LIN {X 0,Y 712.232,Z 484.504,A -85,B 0,C 180,E1 31176.986,E2 31176.986} C_VEL
LIN {X 0,Y 712.279,Z 484.496,A -85,B 0,C 180,E1 31174.064,E2 31174.064} C_VEL
LIN {X 0,Y 712.227,Z 484.507,A -85,B 0,C 180,E1 31171.201,E2 31171.201} C_VEL
LIN {X 0,Y 712.264,Z 484.499,A -85,B 0,C 180,E1 31168.418,E2 31168.418} C_VEL
LIN {X 0,Y 712.248,Z 484.506,A -85,B 0,C 180,E1 31165.352,E2 31165.352} C_VEL
LIN {X 0,Y 712.232,Z 484.504,A -85,B 0,C 180,E1 31162.623,E2 31162.623} C_VEL
LIN {X 0,Y 712.278,Z 484.504,A -85,B 0,C 180,E1 31159.689,E2 31159.689} C_VEL
LIN {X 0,Y 712.231,Z 484.504,A -85,B 0,C 180,E1 31156.81,E2 31156.81} C_VEL
LIN {X 0,Y 712.272,Z 484.5,A -85,B 0,C 180,E1 31153.972,E2 31153.972} C_VEL
LIN {X 0,Y 712.253,Z 484.509,A -85,B 0,C 180,E1 31150.925,E2 31150.925} C_VEL
LIN {X 0,Y 712.246,Z 484.496,A -85,B 0,C 180,E1 31148.07,E2 31148.07} C_VEL
LIN {X 0,Y 712.279,Z 484.51,A -85,B 0,C 180,E1 31145.074,E2 31145.074} C_VEL
LIN {X 0,Y 712.234,Z 484.505,A -85,B 0,C 180,E1 31142.253,E2 31142.253} C_VEL
LIN {X 0,Y 712.282,Z 484.497,A -85,B 0,C 180,E1 31139.437,E2 31139.437} C_VEL
LIN {X 0,Y 712.247,Z 484.508,A -85,B 0,C 180,E1 31136.378,E2 31136.378} C_VEL
LIN {X 0,Y 712.256,Z 484.497,A -85,B 0,C 180,E1 31133.552,E2 31133.552} C_VEL
LIN {X 0,Y 712.274,Z 484.505,A -85,B 0,C 180,E1 31130.465,E2 31130.465} C_VEL
LIN {X 0,Y 712.243,Z 484.503,A -85,B 0,C 180,E1 31127.597,E2 31127.597} C_VEL
LIN {X 0,Y 712.272,Z 484.501,A -85,B 0,C 180,E1 31124.661,E2 31124.661} C_VEL
LIN {X 0,Y 712.243,Z 484.502,A -85,B 0,C 180,E1 31121.756,E2 31121.756} C_VEL
LIN {X 0,Y 712.276,Z 484.497,A -85,B 0,C 180,E1 31120.828,E2 31120.828} C_VEL
LIN {X 0,Y 711.28,Z 484.631,A -85,B 0,C 180,E1 31120.209,E2 31120.209} C_VEL
LIN {X 0,Y 704.888,Z 485.433,A -85,B 0,C 180,E1 31118.473,E2 31118.473} C_VEL
LIN {X 0,Y 704.331,Z 485.495,A -85,B 0,C 180,E1 31118.022,E2 31118.022} C_VEL
LIN {X 0,Y 704.317,Z 485.491,A -85,B 0,C 180,E1 31115.062,E2 31115.062} C_VEL
LIN {X 0,Y 704.34,Z 485.497,A -85,B 0,C 180,E1 31111.973,E2 31111.973} C_VEL
LIN {X 0,Y 704.311,Z 485.491,A -85,B 0,C 180,E1 31109.032,E2 31109.032} C_VEL
LIN {X 0,Y 704.331,Z 485.492,A -85,B 0,C 180,E1 31106.088,E2 31106.088} C_VEL
LIN {X 0,Y 704.307,Z 485.484,A -85,B 0,C 180,E1 31103.194,E2 31103.194} C_VEL
LIN {X 0,Y 704.34,Z 485.487,A -85,B 0,C 180,E1 31100.295,E2 31100.295} C_VEL
LIN {X 0,Y 704.323,Z 485.482,A -85,B 0,C 180,E1 31097.266,E2 31097.266} C_VEL
LIN {X 0,Y 704.337,Z 485.49,A -85,B 0,C 180,E1 31094.301,E2 31094.301} C_VEL
LIN {X 0,Y 704.337,Z 485.5,A -85,B 0,C 180,E1 31091.199,E2 31091.199} C_VEL
LIN {X 0,Y 704.347,Z 485.574,A -85,B 0,C 180,E1 31088.134,E2 31088.134} C_VEL
LIN {X 0,Y 704.441,Z 486.103,A -85,B 0,C 180,E1 31088.022,E2 31088.022} C_VEL
LIN {X 0,Y 711.05,Z 503.243,A -85,B 0,C 180,E1 31086.452,E2 31086.452} C_VEL
LIN {X 0,Y 710.006,Z 548.76,A -85,B 0,C 180,E1 31083.555,E2 31083.555} C_VEL
LIN {X 0,Y 708.985,Z 595.763,A -85,B 0,C 180,E1 31080.65,E2 31080.65} C_VEL
LIN {X 0,Y 708.154,Z 640.537,A -85,B 0,C 180,E1 31077.954,E2 31077.954} C_VEL
LIN {X 0,Y 708.048,Z 651.379,A -85,B 0,C 180,E1 31077.319,E2 31077.319} C_VEL
LIN {X 0,Y 709.566,Z 661.534,A -85,B 0,C 180,E1 31077.131,E2 31077.131} C_VEL
LIN {X 0,Y 708.424,Z 936.016,A -85,B 0,C 180,E1 31074.153,E2 31074.153} C_VEL
LIN {X 0,Y 708.197,Z 963.102,A -85,B 0,C 180,E1 31073.806,E2 31073.806} C_VEL
LIN {X 0,Y 707.957,Z 984.724,A -85,B 0,C 180,E1 31073.382,E2 31073.382} C_VEL
LIN {X 0,Y 707.588,Z 1005.615,A -85,B 0,C 180,E1 31072.823,E2 31072.823} C_VEL
LIN {X 0,Y 707.174,Z 1027.007,A -85,B 0,C 180,E1 31072.092,E2 31072.092} C_VEL
LIN {X 0,Y 706.746,Z 1047.449,A -85,B 0,C 180,E1 31071.234,E2 31071.234} C_VEL
LIN {X 0,Y 706.293,Z 1066.132,A -85,B 0,C 180,E1 31070.294,E2 31070.294} C_VEL
LIN {X 0,Y 705.844,Z 1084.752,A -85,B 0,C 180,E1 31069.186,E2 31069.186} C_VEL
LIN {X 0,Y 705.405,Z 1102.998,A -85,B 0,C 180,E1 31067.913,E2 31067.913} C_VEL
LIN {X 0,Y 705.047,Z 1118.673,A -85,B 0,C 180,E1 31066.646,E2 31066.646} C_VEL
LIN {X 0,Y 704.714,Z 1133.801,A -85,B 0,C 180,E1 31065.217,E2 31065.217} C_VEL
LIN {X 0,Y 704.453,Z 1147.488,A -85,B 0,C 180,E1 31063.711,E2 31063.711} C_VEL
LIN {X 0,Y 704.251,Z 1159.774,A -85,B 0,C 180,E1 31062.129,E2 31062.129} C_VEL
LIN {X 0,Y 704.113,Z 1170.11,A -85,B 0,C 180,E1 31060.555,E2 31060.555} C_VEL
LIN {X 0,Y 704.015,Z 1179.066,A -85,B 0,C 180,E1 31058.905,E2 31058.905} C_VEL
LIN {X 0,Y 703.96,Z 1186.69,A -85,B 0,C 180,E1 31057.18,E2 31057.18} C_VEL
LIN {X 0,Y 703.924,Z 1192.529,A -85,B 0,C 180,E1 31055.461,E2 31055.461} C_VEL
LIN {X 0,Y 703.914,Z 1196.698,A -85,B 0,C 180,E1 31053.746,E2 31053.746} C_VEL
LIN {X 0,Y 703.917,Z 1199.44,A -85,B 0,C 180,E1 31051.954,E2 31051.954} C_VEL
LIN {X 0,Y 703.907,Z 1200.448,A -85,B 0,C 180,E1 31050.163,E2 31050.163} C_VEL
LIN {X 0,Y 703.905,Z 1199.787,A -85,B 0,C 180,E1 31048.372,E2 31048.372} C_VEL
LIN {X 0,Y 703.906,Z 1197.502,A -85,B 0,C 180,E1 31046.58,E2 31046.58} C_VEL
LIN {X 0,Y 703.921,Z 1193.692,A -85,B 0,C 180,E1 31044.866,E2 31044.866} C_VEL
LIN {X 0,Y 703.931,Z 1188.233,A -85,B 0,C 180,E1 31043.148,E2 31043.148} C_VEL
LIN {X 0,Y 703.997,Z 1181.131,A -85,B 0,C 180,E1 31041.424,E2 31041.424} C_VEL
LIN {X 0,Y 704.079,Z 1172.545,A -85,B 0,C 180,E1 31039.775,E2 31039.775} C_VEL
LIN {X 0,Y 704.201,Z 1162.131,A -85,B 0,C 180,E1 31038.119,E2 31038.119} C_VEL
LIN {X 0,Y 704.399,Z 1150.346,A -85,B 0,C 180,E1 31036.539,E2 31036.539} C_VEL
LIN {X 0,Y 704.658,Z 1137.101,A -85,B 0,C 180,E1 31035.034,E2 31035.034} C_VEL
LIN {X 0,Y 704.954,Z 1122.438,A -85,B 0,C 180,E1 31033.606,E2 31033.606} C_VEL
LIN {X 0,Y 705.339,Z 1105.832,A -85,B 0,C 180,E1 31032.213,E2 31032.213} C_VEL
LIN {X 0,Y 705.749,Z 1088.787,A -85,B 0,C 180,E1 31030.983,E2 31030.983} C_VEL
LIN {X 0,Y 706.205,Z 1070.106,A -85,B 0,C 180,E1 31029.838,E2 31029.838} C_VEL
LIN {X 0,Y 706.666,Z 1050.479,A -85,B 0,C 180,E1 31028.82,E2 31028.82} C_VEL
LIN {X 0,Y 707.104,Z 1030.455,A -85,B 0,C 180,E1 31027.95,E2 31027.95} C_VEL
LIN {X 0,Y 707.531,Z 1009.93,A -85,B 0,C 180,E1 31027.219,E2 31027.219} C_VEL
LIN {X 0,Y 707.864,Z 988.627,A -85,B 0,C 180,E1 31026.624,E2 31026.624} C_VEL
LIN {X 0,Y 708.181,Z 965.883,A -85,B 0,C 180,E1 31026.151,E2 31026.151} C_VEL
LIN {X 0,Y 708.392,Z 943.778,A -85,B 0,C 180,E1 31025.841,E2 31025.841} C_VEL
LIN {X 0,Y 709.534,Z 668.723,A -85,B 0,C 180,E1 31022.858,E2 31022.858} C_VEL
LIN {X 0,Y 709.316,Z 658.636,A -85,B 0,C 180,E1 31022.737,E2 31022.737} C_VEL
LIN {X 0,Y 708.045,Z 651.346,A -85,B 0,C 180,E1 31022.59,E2 31022.59} C_VEL
LIN {X 0,Y 708.834,Z 604.03,A -85,B 0,C 180,E1 31019.763,E2 31019.763} C_VEL
LIN {X 0,Y 709.788,Z 557.758,A -85,B 0,C 180,E1 31016.917,E2 31016.917} C_VEL
LIN {X 0,Y 710.872,Z 510.794,A -85,B 0,C 180,E1 31013.945,E2 31013.945} C_VEL
LIN {X 0,Y 710.891,Z 502.371,A -85,B 0,C 180,E1 31013.391,E2 31013.391} C_VEL
LIN {X 0,Y 704.379,Z 485.802,A -85,B 0,C 180,E1 31011.853,E2 31011.853} C_VEL
LIN {X 0,Y 704.318,Z 485.476,A -85,B 0,C 180,E1 31010.927,E2 31010.927} C_VEL
LIN {X 0,Y 704.339,Z 485.484,A -85,B 0,C 180,E1 31007.93,E2 31007.93} C_VEL
LIN {X 0,Y 704.306,Z 485.497,A -85,B 0,C 180,E1 31004.992,E2 31004.992} C_VEL
LIN {X 0,Y 704.332,Z 485.489,A -85,B 0,C 180,E1 31002.072,E2 31002.072} C_VEL
LIN {X 0,Y 704.308,Z 485.49,A -85,B 0,C 180,E1 30999.18,E2 30999.18} C_VEL
LIN {X 0,Y 704.336,Z 485.49,A -85,B 0,C 180,E1 30996.262,E2 30996.262} C_VEL
LIN {X 0,Y 704.322,Z 485.487,A -85,B 0,C 180,E1 30993.229,E2 30993.229} C_VEL
LIN {X 0,Y 704.322,Z 485.497,A -85,B 0,C 180,E1 30990.264,E2 30990.264} C_VEL
LIN {X 0,Y 704.328,Z 485.485,A -85,B 0,C 180,E1 30987.11,E2 30987.11} C_VEL
LIN {X 0,Y 704.309,Z 485.498,A -85,B 0,C 180,E1 30984.223,E2 30984.223} C_VEL
LIN {X 0,Y 704.341,Z 485.49,A -85,B 0,C 180,E1 30981.223,E2 30981.223} C_VEL
LIN {X 0,Y 704.297,Z 485.489,A -85,B 0,C 180,E1 30978.371,E2 30978.371} C_VEL
LIN {X 0,Y 704.34,Z 485.492,A -85,B 0,C 180,E1 30975.479,E2 30975.479} C_VEL
LIN {X 0,Y 704.305,Z 485.492,A -85,B 0,C 180,E1 30972.462,E2 30972.462} C_VEL
LIN {X 0,Y 704.326,Z 485.493,A -85,B 0,C 180,E1 30969.561,E2 30969.561} C_VEL
LIN {X 0,Y 704.313,Z 485.487,A -85,B 0,C 180,E1 30966.418,E2 30966.418} C_VEL
LIN {X 0,Y 704.306,Z 485.497,A -85,B 0,C 180,E1 30963.581,E2 30963.581} C_VEL
LIN {X 0,Y 704.341,Z 485.487,A -85,B 0,C 180,E1 30960.488,E2 30960.488} C_VEL
LIN {X 0,Y 704.292,Z 485.495,A -85,B 0,C 180,E1 30957.64,E2 30957.64} C_VEL
LIN {X 0,Y 704.341,Z 485.497,A -85,B 0,C 180,E1 30954.787,E2 30954.787} C_VEL
LIN {X 0,Y 704.298,Z 485.486,A -85,B 0,C 180,E1 30951.838,E2 30951.838} C_VEL
LIN {X 0,Y 704.314,Z 485.499,A -85,B 0,C 180,E1 30949.033,E2 30949.033} C_VEL
LIN {X 0,Y 704.314,Z 485.491,A -85,B 0,C 180,E1 30945.866,E2 30945.866} C_VEL
LIN {X 0,Y 704.293,Z 485.493,A -85,B 0,C 180,E1 30943.08,E2 30943.08} C_VEL
LIN {X 0,Y 704.342,Z 485.488,A -85,B 0,C 180,E1 30940.08,E2 30940.08} C_VEL
LIN {X 0,Y 704.287,Z 485.495,A -85,B 0,C 180,E1 30937.196,E2 30937.196} C_VEL
LIN {X 0,Y 704.337,Z 485.495,A -85,B 0,C 180,E1 30934.343,E2 30934.343} C_VEL
LIN {X 0,Y 704.298,Z 485.49,A -85,B 0,C 180,E1 30931.323,E2 30931.323} C_VEL
LIN {X 0,Y 704.295,Z 485.497,A -85,B 0,C 180,E1 30928.598,E2 30928.598} C_VEL
LIN {X 0,Y 704.337,Z 485.489,A -85,B 0,C 180,E1 30925.565,E2 30925.565} C_VEL
LIN {X 0,Y 704.283,Z 485.495,A -85,B 0,C 180,E1 30922.785,E2 30922.785} C_VEL
LIN {X 0,Y 704.33,Z 485.484,A -85,B 0,C 180,E1 30919.977,E2 30919.977} C_VEL
LIN {X 0,Y 704.297,Z 485.485,A -85,B 0,C 180,E1 30916.931,E2 30916.931} C_VEL
LIN {X 0,Y 704.29,Z 485.5,A -85,B 0,C 180,E1 30914.191,E2 30914.191} C_VEL
LIN {X 0,Y 704.343,Z 485.487,A -85,B 0,C 180,E1 30911.199,E2 30911.199} C_VEL
LIN {X 0,Y 704.301,Z 485.633,A -85,B 0,C 180,E1 30908.496,E2 30908.496} C_VEL
LIN {X 0,Y 705.145,Z 488.254,A -85,B 0,C 180,E1 30908.226,E2 30908.226} C_VEL
LIN {X 0,Y 711.397,Z 503.301,A -85,B 0,C 180,E1 30906.894,E2 30906.894} C_VEL
LIN {X 0,Y 710.895,Z 527.91,A -85,B 0,C 180,E1 30905.413,E2 30905.413} C_VEL
LIN {X 0,Y 713.276,Z 540.379,A -85,B 0,C 180,E1 30905.117,E2 30905.117} C_VEL
LIN {X 0,Y 711.781,Z 796.504,A -85,B 0,C 180,E1 30902.16,E2 30902.16} C_VEL
LIN {X 0,Y 711.096,Z 919.207,A -85,B 0,C 180,E1 30900.746,E2 30900.746} C_VEL
LIN {X 0,Y 710.67,Z 944.945,A -85,B 0,C 180,E1 30900.302,E2 30900.302} C_VEL
LIN {X 0,Y 710.258,Z 966.602,A -85,B 0,C 180,E1 30899.791,E2 30899.791} C_VEL
LIN {X 0,Y 709.768,Z 990.595,A -85,B 0,C 180,E1 30899.078,E2 30899.078} C_VEL
LIN {X 0,Y 709.163,Z 1012.516,A -85,B 0,C 180,E1 30898.277,E2 30898.277} C_VEL
LIN {X 0,Y 708.561,Z 1035.191,A -85,B 0,C 180,E1 30897.297,E2 30897.297} C_VEL
LIN {X 0,Y 707.882,Z 1056.777,A -85,B 0,C 180,E1 30896.193,E2 30896.193} C_VEL
LIN {X 0,Y 707.236,Z 1077.766,A -85,B 0,C 180,E1 30894.961,E2 30894.961} C_VEL
LIN {X 0,Y 706.625,Z 1097.064,A -85,B 0,C 180,E1 30893.65,E2 30893.65} C_VEL
LIN {X 0,Y 706.064,Z 1115.772,A -85,B 0,C 180,E1 30892.216,E2 30892.216} C_VEL
LIN {X 0,Y 705.557,Z 1132.805,A -85,B 0,C 180,E1 30890.718,E2 30890.718} C_VEL
LIN {X 0,Y 705.141,Z 1148.973,A -85,B 0,C 180,E1 30889.12,E2 30889.12} C_VEL
LIN {X 0,Y 704.767,Z 1163.229,A -85,B 0,C 180,E1 30887.504,E2 30887.504} C_VEL
LIN {X 0,Y 704.49,Z 1177.065,A -85,B 0,C 180,E1 30885.728,E2 30885.728} C_VEL
LIN {X 0,Y 704.267,Z 1188.801,A -85,B 0,C 180,E1 30883.966,E2 30883.966} C_VEL
LIN {X 0,Y 704.115,Z 1198.949,A -85,B 0,C 180,E1 30882.215,E2 30882.215} C_VEL
LIN {X 0,Y 704.003,Z 1208.54,A -85,B 0,C 180,E1 30880.226,E2 30880.226} C_VEL
LIN {X 0,Y 703.953,Z 1215.121,A -85,B 0,C 180,E1 30878.577,E2 30878.577} C_VEL
LIN {X 0,Y 703.926,Z 1221.452,A -85,B 0,C 180,E1 30876.607,E2 30876.607} C_VEL
LIN {X 0,Y 703.911,Z 1225.814,A -85,B 0,C 180,E1 30874.726,E2 30874.726} C_VEL
LIN {X 0,Y 703.882,Z 1228.685,A -85,B 0,C 180,E1 30872.931,E2 30872.931} C_VEL
LIN {X 0,Y 703.892,Z 1230.262,A -85,B 0,C 180,E1 30870.895,E2 30870.895} C_VEL
LIN {X 0,Y 703.884,Z 1230.306,A -85,B 0,C 180,E1 30869.267,E2 30869.267} C_VEL
LIN {X 0,Y 703.886,Z 1229.017,A -85,B 0,C 180,E1 30867.313,E2 30867.313} C_VEL
LIN {X 0,Y 703.916,Z 1225.973,A -85,B 0,C 180,E1 30865.356,E2 30865.356} C_VEL
LIN {X 0,Y 703.925,Z 1221.865,A -85,B 0,C 180,E1 30863.557,E2 30863.557} C_VEL
LIN {X 0,Y 703.956,Z 1215.424,A -85,B 0,C 180,E1 30861.505,E2 30861.505} C_VEL
LIN {X 0,Y 703.996,Z 1208.765,A -85,B 0,C 180,E1 30859.826,E2 30859.826} C_VEL
LIN {X 0,Y 704.106,Z 1199.868,A -85,B 0,C 180,E1 30857.951,E2 30857.951} C_VEL
LIN {X 0,Y 704.26,Z 1189.323,A -85,B 0,C 180,E1 30856.117,E2 30856.117} C_VEL
LIN {X 0,Y 704.473,Z 1177.647,A -85,B 0,C 180,E1 30854.356,E2 30854.356} C_VEL
LIN {X 0,Y 704.749,Z 1163.936,A -85,B 0,C 180,E1 30852.581,E2 30852.581} C_VEL
LIN {X 0,Y 705.119,Z 1149.75,A -85,B 0,C 180,E1 30850.965,E2 30850.965} C_VEL
LIN {X 0,Y 705.54,Z 1133.398,A -85,B 0,C 180,E1 30849.337,E2 30849.337} C_VEL
LIN {X 0,Y 706.035,Z 1116.552,A -85,B 0,C 180,E1 30847.85,E2 30847.85} C_VEL
LIN {X 0,Y 706.604,Z 1097.667,A -85,B 0,C 180,E1 30846.394,E2 30846.394} C_VEL
LIN {X 0,Y 707.213,Z 1078.429,A -85,B 0,C 180,E1 30845.083,E2 30845.083} C_VEL
LIN {X 0,Y 707.852,Z 1057.575,A -85,B 0,C 180,E1 30843.851,E2 30843.851} C_VEL
LIN {X 0,Y 708.498,Z 1036.993,A -85,B 0,C 180,E1 30842.791,E2 30842.791} C_VEL
LIN {X 0,Y 709.128,Z 1013.638,A -85,B 0,C 180,E1 30841.768,E2 30841.768} C_VEL
LIN {X 0,Y 709.724,Z 991.879,A -85,B 0,C 180,E1 30840.966,E2 30840.966} C_VEL
LIN {X 0,Y 710.256,Z 966.819,A -85,B 0,C 180,E1 30840.214,E2 30840.214} C_VEL
LIN {X 0,Y 710.662,Z 945.208,A -85,B 0,C 180,E1 30839.704,E2 30839.704} C_VEL
LIN {X 0,Y 711.094,Z 919.454,A -85,B 0,C 180,E1 30839.258,E2 30839.258} C_VEL
LIN {X 0,Y 711.703,Z 811.771,A -85,B 0,C 180,E1 30838.014,E2 30838.014} C_VEL
LIN {X 0,Y 713.129,Z 564.423,A -85,B 0,C 180,E1 30835.164,E2 30835.164} C_VEL
LIN {X 0,Y 713.107,Z 538.54,A -85,B 0,C 180,E1 30834.851,E2 30834.851} C_VEL
LIN {X 0,Y 710.908,Z 527.965,A -85,B 0,C 180,E1 30834.588,E2 30834.588} C_VEL
LIN {X 0,Y 711.397,Z 503.3,A -85,B 0,C 180,E1 30833.106,E2 30833.106} C_VEL
LIN {X 0,Y 704.326,Z 485.803,A -85,B 0,C 180,E1 30831.541,E2 30831.541} C_VEL
LIN {X 0,Y 704.342,Z 485.485,A -85,B 0,C 180,E1 30830.558,E2 30830.558} C_VEL
LIN {X 0,Y 704.281,Z 485.485,A -85,B 0,C 180,E1 30827.705,E2 30827.705} C_VEL
LIN {X 0,Y 704.312,Z 485.494,A -85,B 0,C 180,E1 30824.991,E2 30824.991} C_VEL
LIN {X 0,Y 704.307,Z 485.5,A -85,B 0,C 180,E1 30821.855,E2 30821.855} C_VEL
LIN {X 0,Y 704.284,Z 485.478,A -85,B 0,C 180,E1 30819.182,E2 30819.182} C_VEL
LIN {X 0,Y 704.341,Z 485.495,A -85,B 0,C 180,E1 30816.263,E2 30816.263} C_VEL
LIN {X 0,Y 704.289,Z 485.482,A -85,B 0,C 180,E1 30813.328,E2 30813.328} C_VEL
LIN {X 0,Y 704.317,Z 485.491,A -85,B 0,C 180,E1 30810.547,E2 30810.547} C_VEL
LIN {X 0,Y 704.315,Z 485.5,A -85,B 0,C 180,E1 30807.469,E2 30807.469} C_VEL
LIN {X 0,Y 704.294,Z 485.489,A -85,B 0,C 180,E1 30804.67,E2 30804.67} C_VEL
LIN {X 0,Y 704.341,Z 485.496,A -85,B 0,C 180,E1 30801.748,E2 30801.748} C_VEL
LIN {X 0,Y 704.292,Z 485.496,A -85,B 0,C 180,E1 30798.887,E2 30798.887} C_VEL
LIN {X 0,Y 704.33,Z 485.486,A -85,B 0,C 180,E1 30796.042,E2 30796.042} C_VEL
LIN {X 0,Y 704.311,Z 485.493,A -85,B 0,C 180,E1 30792.962,E2 30792.962} C_VEL
LIN {X 0,Y 704.306,Z 485.491,A -85,B 0,C 180,E1 30790.139,E2 30790.139} C_VEL
LIN {X 0,Y 704.343,Z 485.493,A -85,B 0,C 180,E1 30787.095,E2 30787.095} C_VEL
LIN {X 0,Y 704.295,Z 485.489,A -85,B 0,C 180,E1 30784.234,E2 30784.234} C_VEL
LIN {X 0,Y 704.34,Z 485.49,A -85,B 0,C 180,E1 30781.383,E2 30781.383} C_VEL
LIN {X 0,Y 704.309,Z 485.496,A -85,B 0,C 180,E1 30778.454,E2 30778.454} C_VEL
LIN {X 0,Y 704.319,Z 485.489,A -85,B 0,C 180,E1 30775.603,E2 30775.603} C_VEL
LIN {X 0,Y 704.333,Z 485.5,A -85,B 0,C 180,E1 30772.495,E2 30772.495} C_VEL
LIN {X 0,Y 704.306,Z 485.485,A -85,B 0,C 180,E1 30769.613,E2 30769.613} C_VEL
LIN {X 0,Y 704.337,Z 485.497,A -85,B 0,C 180,E1 30766.621,E2 30766.621} C_VEL
LIN {X 0,Y 704.301,Z 485.495,A -85,B 0,C 180,E1 30763.759,E2 30763.759} C_VEL
LIN {X 0,Y 704.339,Z 485.485,A -85,B 0,C 180,E1 30760.857,E2 30760.857} C_VEL
LIN {X 0,Y 704.331,Z 485.495,A -85,B 0,C 180,E1 30758.022,E2 30758.022} C_VEL
LIN {X 0,Y 703.303,Z 485.614,A -85,B 0,C 180,E1 30757.395,E2 30757.395} C_VEL
LIN {X 0,Y 696.884,Z 486.424,A -85,B 0,C 180,E1 30755.639,E2 30755.639} C_VEL
LIN {X 0,Y 696.37,Z 486.481,A -85,B 0,C 180,E1 30755.183,E2 30755.183} C_VEL
LIN {X 0,Y 696.396,Z 486.481,A -85,B 0,C 180,E1 30752.181,E2 30752.181} C_VEL
LIN {X 0,Y 696.368,Z 486.484,A -85,B 0,C 180,E1 30749.323,E2 30749.323} C_VEL
LIN {X 0,Y 696.398,Z 486.476,A -85,B 0,C 180,E1 30746.381,E2 30746.381} C_VEL
LIN {X 0,Y 696.378,Z 486.473,A -85,B 0,C 180,E1 30743.38,E2 30743.38} C_VEL
LIN {X 0,Y 696.402,Z 486.475,A -85,B 0,C 180,E1 30740.395,E2 30740.395} C_VEL
LIN {X 0,Y 696.389,Z 486.468,A -85,B 0,C 180,E1 30737.317,E2 30737.317} C_VEL
LIN {X 0,Y 696.4,Z 486.479,A -85,B 0,C 180,E1 30734.249,E2 30734.249} C_VEL
LIN {X 0,Y 696.391,Z 486.489,A -85,B 0,C 180,E1 30731.116,E2 30731.116} C_VEL
LIN {X 0,Y 696.399,Z 486.668,A -85,B 0,C 180,E1 30728.527,E2 30728.527} C_VEL
LIN {X 0,Y 700.012,Z 495.946,A -85,B 0,C 180,E1 30727.623,E2 30727.623} C_VEL
LIN {X 0,Y 704.1,Z 506.677,A -85,B 0,C 180,E1 30726.644,E2 30726.644} C_VEL
LIN {X 0,Y 702.908,Z 551.847,A -85,B 0,C 180,E1 30723.743,E2 30723.743} C_VEL
LIN {X 0,Y 701.724,Z 599.512,A -85,B 0,C 180,E1 30720.771,E2 30720.771} C_VEL
LIN {X 0,Y 700.761,Z 644.343,A -85,B 0,C 180,E1 30718.043,E2 30718.043} C_VEL
LIN {X 0,Y 700.767,Z 651.94,A -85,B 0,C 180,E1 30717.615,E2 30717.615} C_VEL
LIN {X 0,Y 702.441,Z 662.731,A -85,B 0,C 180,E1 30717.416,E2 30717.416} C_VEL
LIN {X 0,Y 701.12,Z 937.085,A -85,B 0,C 180,E1 30714.409,E2 30714.409} C_VEL
LIN {X 0,Y 700.865,Z 963.369,A -85,B 0,C 180,E1 30714.067,E2 30714.067} C_VEL
LIN {X 0,Y 700.585,Z 984.94,A -85,B 0,C 180,E1 30713.638,E2 30713.638} C_VEL
LIN {X 0,Y 700.158,Z 1006.371,A -85,B 0,C 180,E1 30713.057,E2 30713.057} C_VEL
LIN {X 0,Y 699.698,Z 1027.018,A -85,B 0,C 180,E1 30712.34,E2 30712.34} C_VEL
LIN {X 0,Y 699.197,Z 1047.457,A -85,B 0,C 180,E1 30711.474,E2 30711.474} C_VEL
LIN {X 0,Y 698.68,Z 1066.146,A -85,B 0,C 180,E1 30710.525,E2 30710.525} C_VEL
LIN {X 0,Y 698.165,Z 1084.759,A -85,B 0,C 180,E1 30709.405,E2 30709.405} C_VEL
LIN {X 0,Y 697.651,Z 1103.003,A -85,B 0,C 180,E1 30708.119,E2 30708.119} C_VEL
LIN {X 0,Y 697.233,Z 1118.679,A -85,B 0,C 180,E1 30706.838,E2 30706.838} C_VEL
LIN {X 0,Y 696.845,Z 1134.062,A -85,B 0,C 180,E1 30705.367,E2 30705.367} C_VEL
LIN {X 0,Y 696.548,Z 1147.492,A -85,B 0,C 180,E1 30703.87,E2 30703.87} C_VEL
LIN {X 0,Y 696.313,Z 1159.779,A -85,B 0,C 180,E1 30702.27,E2 30702.27} C_VEL
LIN {X 0,Y 696.145,Z 1170.112,A -85,B 0,C 180,E1 30700.677,E2 30700.677} C_VEL
LIN {X 0,Y 696.03,Z 1179.069,A -85,B 0,C 180,E1 30699.008,E2 30699.008} C_VEL
LIN {X 0,Y 695.967,Z 1186.692,A -85,B 0,C 180,E1 30697.263,E2 30697.263} C_VEL
LIN {X 0,Y 695.923,Z 1192.531,A -85,B 0,C 180,E1 30695.524,E2 30695.524} C_VEL
LIN {X 0,Y 695.915,Z 1196.699,A -85,B 0,C 180,E1 30693.789,E2 30693.789} C_VEL
LIN {X 0,Y 695.917,Z 1199.44,A -85,B 0,C 180,E1 30691.976,E2 30691.976} C_VEL
LIN {X 0,Y 695.907,Z 1200.448,A -85,B 0,C 180,E1 30690.165,E2 30690.165} C_VEL
LIN {X 0,Y 695.906,Z 1199.787,A -85,B 0,C 180,E1 30688.353,E2 30688.353} C_VEL
LIN {X 0,Y 695.909,Z 1197.501,A -85,B 0,C 180,E1 30686.54,E2 30686.54} C_VEL
LIN {X 0,Y 695.924,Z 1193.69,A -85,B 0,C 180,E1 30684.807,E2 30684.807} C_VEL
LIN {X 0,Y 695.94,Z 1188.232,A -85,B 0,C 180,E1 30683.069,E2 30683.069} C_VEL
LIN {X 0,Y 696.011,Z 1181.129,A -85,B 0,C 180,E1 30681.325,E2 30681.325} C_VEL
LIN {X 0,Y 696.11,Z 1172.543,A -85,B 0,C 180,E1 30679.657,E2 30679.657} C_VEL
LIN {X 0,Y 696.261,Z 1161.937,A -85,B 0,C 180,E1 30677.954,E2 30677.954} C_VEL
LIN {X 0,Y 696.484,Z 1150.341,A -85,B 0,C 180,E1 30676.383,E2 30676.383} C_VEL
LIN {X 0,Y 696.783,Z 1137.097,A -85,B 0,C 180,E1 30674.861,E2 30674.861} C_VEL
LIN {X 0,Y 697.134,Z 1122.431,A -85,B 0,C 180,E1 30673.416,E2 30673.416} C_VEL
LIN {X 0,Y 697.579,Z 1105.826,A -85,B 0,C 180,E1 30672.008,E2 30672.008} C_VEL
LIN {X 0,Y 698.052,Z 1088.782,A -85,B 0,C 180,E1 30670.765,E2 30670.765} C_VEL
LIN {X 0,Y 698.558,Z 1070.703,A -85,B 0,C 180,E1 30669.644,E2 30669.644} C_VEL
LIN {X 0,Y 699.095,Z 1051.047,A -85,B 0,C 180,E1 30668.608,E2 30668.608} C_VEL
LIN {X 0,Y 699.593,Z 1031.566,A -85,B 0,C 180,E1 30667.745,E2 30667.745} C_VEL
LIN {X 0,Y 700.066,Z 1011.197,A -85,B 0,C 180,E1 30667.007,E2 30667.007} C_VEL
LIN {X 0,Y 700.47,Z 989.6,A -85,B 0,C 180,E1 30666.388,E2 30666.388} C_VEL
LIN {X 0,Y 700.836,Z 967.551,A -85,B 0,C 180,E1 30665.914,E2 30665.914} C_VEL
LIN {X 0,Y 701.068,Z 945.826,A -85,B 0,C 180,E1 30665.597,E2 30665.597} C_VEL
LIN {X 0,Y 702.393,Z 672.108,A -85,B 0,C 180,E1 30662.598,E2 30662.598} C_VEL
LIN {X 0,Y 702.203,Z 659.929,A -85,B 0,C 180,E1 30662.452,E2 30662.452} C_VEL
LIN {X 0,Y 700.694,Z 651.352,A -85,B 0,C 180,E1 30662.278,E2 30662.278} C_VEL
LIN {X 0,Y 701.612,Z 604.826,A -85,B 0,C 180,E1 30659.466,E2 30659.466} C_VEL
LIN {X 0,Y 702.741,Z 557.792,A -85,B 0,C 180,E1 30656.542,E2 30656.542} C_VEL
LIN {X 0,Y 703.968,Z 511.51,A -85,B 0,C 180,E1 30653.581,E2 30653.581} C_VEL
LIN {X 0,Y 704.051,Z 506.113,A -85,B 0,C 180,E1 30653.225,E2 30653.225} C_VEL
LIN {X 0,Y 696.401,Z 486.723,A -85,B 0,C 180,E1 30651.39,E2 30651.39} C_VEL
LIN {X 0,Y 696.39,Z 486.49,A -85,B 0,C 180,E1 30648.775,E2 30648.775} C_VEL
LIN {X 0,Y 696.391,Z 486.48,A -85,B 0,C 180,E1 30645.636,E2 30645.636} C_VEL
LIN {X 0,Y 696.38,Z 486.469,A -85,B 0,C 180,E1 30642.666,E2 30642.666} C_VEL
LIN {X 0,Y 696.399,Z 486.476,A -85,B 0,C 180,E1 30639.556,E2 30639.556} C_VEL
LIN {X 0,Y 696.372,Z 486.473,A -85,B 0,C 180,E1 30636.576,E2 30636.576} C_VEL
LIN {X 0,Y 696.402,Z 486.476,A -85,B 0,C 180,E1 30633.558,E2 30633.558} C_VEL
LIN {X 0,Y 696.363,Z 486.484,A -85,B 0,C 180,E1 30630.646,E2 30630.646} C_VEL
LIN {X 0,Y 696.4,Z 486.482,A -85,B 0,C 180,E1 30627.816,E2 30627.816} C_VEL
LIN {X 0,Y 696.366,Z 486.482,A -85,B 0,C 180,E1 30624.789,E2 30624.789} C_VEL
LIN {X 0,Y 696.401,Z 486.484,A -85,B 0,C 180,E1 30621.831,E2 30621.831} C_VEL
LIN {X 0,Y 696.376,Z 486.474,A -85,B 0,C 180,E1 30618.762,E2 30618.762} C_VEL
LIN {X 0,Y 696.38,Z 486.488,A -85,B 0,C 180,E1 30615.832,E2 30615.832} C_VEL
LIN {X 0,Y 696.386,Z 486.479,A -85,B 0,C 180,E1 30612.69,E2 30612.69} C_VEL
LIN {X 0,Y 696.364,Z 486.479,A -85,B 0,C 180,E1 30609.838,E2 30609.838} C_VEL
LIN {X 0,Y 696.401,Z 486.475,A -85,B 0,C 180,E1 30606.844,E2 30606.844} C_VEL
LIN {X 0,Y 696.354,Z 486.483,A -85,B 0,C 180,E1 30603.952,E2 30603.952} C_VEL
LIN {X 0,Y 696.404,Z 486.48,A -85,B 0,C 180,E1 30601.07,E2 30601.07} C_VEL
LIN {X 0,Y 696.367,Z 486.48,A -85,B 0,C 180,E1 30598.107,E2 30598.107} C_VEL
LIN {X 0,Y 696.368,Z 486.482,A -85,B 0,C 180,E1 30595.305,E2 30595.305} C_VEL
LIN {X 0,Y 696.391,Z 486.471,A -85,B 0,C 180,E1 30592.171,E2 30592.171} C_VEL
LIN {X 0,Y 696.355,Z 486.486,A -85,B 0,C 180,E1 30589.325,E2 30589.325} C_VEL
LIN {X 0,Y 696.401,Z 486.483,A -85,B 0,C 180,E1 30586.381,E2 30586.381} C_VEL
LIN {X 0,Y 696.351,Z 486.479,A -85,B 0,C 180,E1 30583.482,E2 30583.482} C_VEL
LIN {X 0,Y 696.39,Z 486.489,A -85,B 0,C 180,E1 30580.629,E2 30580.629} C_VEL
LIN {X 0,Y 696.365,Z 486.481,A -85,B 0,C 180,E1 30577.546,E2 30577.546} C_VEL
LIN {X 0,Y 696.358,Z 486.482,A -85,B 0,C 180,E1 30574.757,E2 30574.757} C_VEL
LIN {X 0,Y 696.397,Z 486.476,A -85,B 0,C 180,E1 30571.657,E2 30571.657} C_VEL
LIN {X 0,Y 696.347,Z 486.484,A -85,B 0,C 180,E1 30568.845,E2 30568.845} C_VEL
LIN {X 0,Y 696.401,Z 486.469,A -85,B 0,C 180,E1 30565.937,E2 30565.937} C_VEL
LIN {X 0,Y 696.352,Z 486.483,A -85,B 0,C 180,E1 30562.971,E2 30562.971} C_VEL
LIN {X 0,Y 696.357,Z 486.468,A -85,B 0,C 180,E1 30560.285,E2 30560.285} C_VEL
LIN {X 0,Y 696.386,Z 486.471,A -85,B 0,C 180,E1 30557.196,E2 30557.196} C_VEL
LIN {X 0,Y 696.344,Z 486.488,A -85,B 0,C 180,E1 30554.368,E2 30554.368} C_VEL
LIN {X 0,Y 696.403,Z 486.469,A -85,B 0,C 180,E1 30551.443,E2 30551.443} C_VEL
LIN {X 0,Y 696.403,Z 486.623,A -85,B 0,C 180,E1 30548.939,E2 30548.939} C_VEL
LIN {X 0,Y 697.498,Z 489.736,A -85,B 0,C 180,E1 30548.622,E2 30548.622} C_VEL
LIN {X 0,Y 704.529,Z 506.76,A -85,B 0,C 180,E1 30547.096,E2 30547.096} C_VEL
LIN {X 0,Y 704.075,Z 528.398,A -85,B 0,C 180,E1 30545.798,E2 30545.798} C_VEL
LIN {X 0,Y 706.716,Z 541.979,A -85,B 0,C 180,E1 30545.473,E2 30545.473} C_VEL
LIN {X 0,Y 704.999,Z 797.522,A -85,B 0,C 180,E1 30542.495,E2 30542.495} C_VEL
LIN {X 0,Y 704.211,Z 919.325,A -85,B 0,C 180,E1 30541.078,E2 30541.078} C_VEL
LIN {X 0,Y 703.739,Z 944.943,A -85,B 0,C 180,E1 30540.632,E2 30540.632} C_VEL
LIN {X 0,Y 703.251,Z 966.713,A -85,B 0,C 180,E1 30540.116,E2 30540.116} C_VEL
LIN {X 0,Y 702.691,Z 990.591,A -85,B 0,C 180,E1 30539.4,E2 30539.4} C_VEL
LIN {X 0,Y 702.01,Z 1012.515,A -85,B 0,C 180,E1 30538.591,E2 30538.591} C_VEL
LIN {X 0,Y 701.294,Z 1035.187,A -85,B 0,C 180,E1 30537.604,E2 30537.604} C_VEL
LIN {X 0,Y 700.539,Z 1056.573,A -85,B 0,C 180,E1 30536.5,E2 30536.5} C_VEL
LIN {X 0,Y 699.774,Z 1077.76,A -85,B 0,C 180,E1 30535.246,E2 30535.246} C_VEL
LIN {X 0,Y 699.093,Z 1096.755,A -85,B 0,C 180,E1 30533.943,E2 30533.943} C_VEL
LIN {X 0,Y 698.419,Z 1115.771,A -85,B 0,C 180,E1 30532.472,E2 30532.472} C_VEL
LIN {X 0,Y 697.846,Z 1132.471,A -85,B 0,C 180,E1 30530.989,E2 30530.989} C_VEL
LIN {X 0,Y 697.345,Z 1148.975,A -85,B 0,C 180,E1 30529.342,E2 30529.342} C_VEL
LIN {X 0,Y 696.901,Z 1163.938,A -85,B 0,C 180,E1 30527.621,E2 30527.621} C_VEL
LIN {X 0,Y 696.576,Z 1177.648,A -85,B 0,C 180,E1 30525.826,E2 30525.826} C_VEL
LIN {X 0,Y 696.321,Z 1189.322,A -85,B 0,C 180,E1 30524.044,E2 30524.044} C_VEL
LIN {X 0,Y 696.136,Z 1200.301,A -85,B 0,C 180,E1 30522.105,E2 30522.105} C_VEL
LIN {X 0,Y 696.017,Z 1208.98,A -85,B 0,C 180,E1 30520.241,E2 30520.241} C_VEL
LIN {X 0,Y 695.963,Z 1215.728,A -85,B 0,C 180,E1 30518.51,E2 30518.51} C_VEL
LIN {X 0,Y 695.927,Z 1222.071,A -85,B 0,C 180,E1 30516.434,E2 30516.434} C_VEL
LIN {X 0,Y 695.913,Z 1225.973,A -85,B 0,C 180,E1 30514.697,E2 30514.697} C_VEL
LIN {X 0,Y 695.883,Z 1228.91,A -85,B 0,C 180,E1 30512.8,E2 30512.8} C_VEL
LIN {X 0,Y 695.888,Z 1230.284,A -85,B 0,C 180,E1 30510.823,E2 30510.823} C_VEL
LIN {X 0,Y 695.888,Z 1230.284,A -85,B 0,C 180,E1 30509.177,E2 30509.177} C_VEL
LIN {X 0,Y 695.883,Z 1228.91,A -85,B 0,C 180,E1 30507.2,E2 30507.2} C_VEL
LIN {X 0,Y 695.913,Z 1225.973,A -85,B 0,C 180,E1 30505.302,E2 30505.302} C_VEL
LIN {X 0,Y 695.928,Z 1221.864,A -85,B 0,C 180,E1 30503.483,E2 30503.483} C_VEL
LIN {X 0,Y 695.96,Z 1215.424,A -85,B 0,C 180,E1 30501.407,E2 30501.407} C_VEL
LIN {X 0,Y 696.02,Z 1208.895,A -85,B 0,C 180,E1 30499.739,E2 30499.739} C_VEL
LIN {X 0,Y 696.143,Z 1199.866,A -85,B 0,C 180,E1 30497.811,E2 30497.811} C_VEL
LIN {X 0,Y 696.321,Z 1189.324,A -85,B 0,C 180,E1 30495.956,E2 30495.956} C_VEL
LIN {X 0,Y 696.593,Z 1177.122,A -85,B 0,C 180,E1 30494.096,E2 30494.096} C_VEL
LIN {X 0,Y 696.923,Z 1163.231,A -85,B 0,C 180,E1 30492.293,E2 30492.293} C_VEL
LIN {X 0,Y 697.369,Z 1148.181,A -85,B 0,C 180,E1 30490.571,E2 30490.571} C_VEL
LIN {X 0,Y 697.875,Z 1131.542,A -85,B 0,C 180,E1 30488.924,E2 30488.924} C_VEL
LIN {X 0,Y 698.487,Z 1113.618,A -85,B 0,C 180,E1 30487.352,E2 30487.352} C_VEL
LIN {X 0,Y 699.129,Z 1095.654,A -85,B 0,C 180,E1 30485.977,E2 30485.977} C_VEL
LIN {X 0,Y 699.843,Z 1075.64,A -85,B 0,C 180,E1 30484.621,E2 30484.621} C_VEL
LIN {X 0,Y 700.56,Z 1055.965,A -85,B 0,C 180,E1 30483.467,E2 30483.467} C_VEL
LIN {X 0,Y 701.325,Z 1034.264,A -85,B 0,C 180,E1 30482.351,E2 30482.351} C_VEL
LIN {X 0,Y 702.011,Z 1012.517,A -85,B 0,C 180,E1 30481.409,E2 30481.409} C_VEL
LIN {X 0,Y 702.717,Z 989.858,A -85,B 0,C 180,E1 30480.575,E2 30480.575} C_VEL
LIN {X 0,Y 703.267,Z 965.653,A -85,B 0,C 180,E1 30479.856,E2 30479.856} C_VEL
LIN {X 0,Y 703.791,Z 943.382,A -85,B 0,C 180,E1 30479.335,E2 30479.335} C_VEL
LIN {X 0,Y 704.219,Z 918.029,A -85,B 0,C 180,E1 30478.904,E2 30478.904} C_VEL
LIN {X 0,Y 705.855,Z 661.925,A -85,B 0,C 180,E1 30475.933,E2 30475.933} C_VEL
LIN {X 0,Y 706.555,Z 540.21,A -85,B 0,C 180,E1 30474.496,E2 30474.496} C_VEL
LIN {X 0,Y 704.009,Z 527.936,A -85,B 0,C 180,E1 30474.187,E2 30474.187} C_VEL
LIN {X 0,Y 704.529,Z 506.741,A -85,B 0,C 180,E1 30472.903,E2 30472.903} C_VEL
LIN {X 0,Y 696.424,Z 486.787,A -85,B 0,C 180,E1 30471.094,E2 30471.094} C_VEL
LIN {X 0,Y 696.384,Z 486.478,A -85,B 0,C 180,E1 30470.288,E2 30470.288} C_VEL
LIN {X 0,Y 696.341,Z 486.473,A -85,B 0,C 180,E1 30467.557,E2 30467.557} C_VEL
LIN {X 0,Y 696.4,Z 486.476,A -85,B 0,C 180,E1 30464.708,E2 30464.708} C_VEL
LIN {X 0,Y 696.352,Z 486.489,A -85,B 0,C 180,E1 30461.669,E2 30461.669} C_VEL
LIN {X 0,Y 696.362,Z 486.462,A -85,B 0,C 180,E1 30458.902,E2 30458.902} C_VEL
LIN {X 0,Y 696.378,Z 486.485,A -85,B 0,C 180,E1 30455.76,E2 30455.76} C_VEL
LIN {X 0,Y 696.349,Z 486.467,A -85,B 0,C 180,E1 30452.971,E2 30452.971} C_VEL
LIN {X 0,Y 696.404,Z 486.484,A -85,B 0,C 180,E1 30450.031,E2 30450.031} C_VEL
LIN {X 0,Y 696.355,Z 486.486,A -85,B 0,C 180,E1 30447.169,E2 30447.169} C_VEL
LIN {X 0,Y 696.384,Z 486.475,A -85,B 0,C 180,E1 30444.336,E2 30444.336} C_VEL
LIN {X 0,Y 696.37,Z 486.483,A -85,B 0,C 180,E1 30441.213,E2 30441.213} C_VEL
LIN {X 0,Y 696.365,Z 486.481,A -85,B 0,C 180,E1 30438.364,E2 30438.364} C_VEL
LIN {X 0,Y 696.395,Z 486.489,A -85,B 0,C 180,E1 30435.241,E2 30435.241} C_VEL
LIN {X 0,Y 696.355,Z 486.477,A -85,B 0,C 180,E1 30432.438,E2 30432.438} C_VEL
LIN {X 0,Y 696.399,Z 486.482,A -85,B 0,C 180,E1 30429.504,E2 30429.504} C_VEL
LIN {X 0,Y 696.361,Z 486.485,A -85,B 0,C 180,E1 30426.596,E2 30426.596} C_VEL
LIN {X 0,Y 696.391,Z 486.473,A -85,B 0,C 180,E1 30423.705,E2 30423.705} C_VEL
LIN {X 0,Y 696.375,Z 486.484,A -85,B 0,C 180,E1 30420.576,E2 30420.576} C_VEL
LIN {X 0,Y 696.376,Z 486.477,A -85,B 0,C 180,E1 30417.696,E2 30417.696} C_VEL
LIN {X 0,Y 696.392,Z 486.481,A -85,B 0,C 180,E1 30414.562,E2 30414.562} C_VEL
LIN {X 0,Y 696.368,Z 486.481,A -85,B 0,C 180,E1 30411.661,E2 30411.661} C_VEL
LIN {X 0,Y 696.399,Z 486.479,A -85,B 0,C 180,E1 30408.656,E2 30408.656} C_VEL
LIN {X 0,Y 696.36,Z 486.477,A -85,B 0,C 180,E1 30405.739,E2 30405.739} C_VEL
LIN {X 0,Y 696.4,Z 486.479,A -85,B 0,C 180,E1 30402.882,E2 30402.882} C_VEL
LIN {X 0,Y 696.372,Z 486.486,A -85,B 0,C 180,E1 30399.842,E2 30399.842} C_VEL
LIN {X 0,Y 696.397,Z 486.472,A -85,B 0,C 180,E1 30396.922,E2 30396.922} C_VEL
LIN {X 0,Y 696.37,Z 486.481,A -85,B 0,C 180,E1 30395.183,E2 30395.183} C_VEL
LIN {X 0,Y 695.404,Z 486.605,A -85,B 0,C 180,E1 30394.549,E2 30394.549} C_VEL
LIN {X 0,Y 688.991,Z 487.397,A -85,B 0,C 180,E1 30392.773,E2 30392.773} C_VEL
LIN {X 0,Y 688.455,Z 487.468,A -85,B 0,C 180,E1 30392.312,E2 30392.312} C_VEL
LIN {X 0,Y 688.434,Z 487.474,A -85,B 0,C 180,E1 30389.446,E2 30389.446} C_VEL
LIN {X 0,Y 688.461,Z 487.464,A -85,B 0,C 180,E1 30386.473,E2 30386.473} C_VEL
LIN {X 0,Y 688.441,Z 487.461,A -85,B 0,C 180,E1 30383.432,E2 30383.432} C_VEL
LIN {X 0,Y 688.463,Z 487.465,A -85,B 0,C 180,E1 30380.388,E2 30380.388} C_VEL
LIN {X 0,Y 688.447,Z 487.455,A -85,B 0,C 180,E1 30377.292,E2 30377.292} C_VEL
LIN {X 0,Y 688.46,Z 487.469,A -85,B 0,C 180,E1 30374.273,E2 30374.273} C_VEL
LIN {X 0,Y 688.455,Z 487.479,A -85,B 0,C 180,E1 30371.14,E2 30371.14} C_VEL
LIN {X 0,Y 688.47,Z 487.65,A -85,B 0,C 180,E1 30368.987,E2 30368.987} C_VEL
LIN {X 0,Y 692.113,Z 496.984,A -85,B 0,C 180,E1 30368.06,E2 30368.06} C_VEL
LIN {X 0,Y 697.153,Z 510.211,A -85,B 0,C 180,E1 30366.834,E2 30366.834} C_VEL
LIN {X 0,Y 695.787,Z 555.692,A -85,B 0,C 180,E1 30363.887,E2 30363.887} C_VEL
LIN {X 0,Y 694.465,Z 603.265,A -85,B 0,C 180,E1 30360.893,E2 30360.893} C_VEL
LIN {X 0,Y 693.353,Z 648.989,A -85,B 0,C 180,E1 30358.084,E2 30358.084} C_VEL
LIN {X 0,Y 693.49,Z 652.059,A -85,B 0,C 180,E1 30357.939,E2 30357.939} C_VEL
LIN {X 0,Y 695.333,Z 663.927,A -85,B 0,C 180,E1 30357.707,E2 30357.707} C_VEL
LIN {X 0,Y 693.832,Z 937.9,A -85,B 0,C 180,E1 30354.674,E2 30354.674} C_VEL
LIN {X 0,Y 693.548,Z 963.443,A -85,B 0,C 180,E1 30354.336,E2 30354.336} C_VEL
LIN {X 0,Y 693.226,Z 985.226,A -85,B 0,C 180,E1 30353.897,E2 30353.897} C_VEL
LIN {X 0,Y 692.75,Z 1006.392,A -85,B 0,C 180,E1 30353.318,E2 30353.318} C_VEL
LIN {X 0,Y 692.235,Z 1027.029,A -85,B 0,C 180,E1 30352.595,E2 30352.595} C_VEL
LIN {X 0,Y 691.688,Z 1046.565,A -85,B 0,C 180,E1 30351.764,E2 30351.764} C_VEL
LIN {X 0,Y 691.107,Z 1065.357,A -85,B 0,C 180,E1 30350.804,E2 30350.804} C_VEL
LIN {X 0,Y 690.514,Z 1084.095,A -85,B 0,C 180,E1 30349.673,E2 30349.673} C_VEL
LIN {X 0,Y 689.941,Z 1101.899,A -85,B 0,C 180,E1 30348.417,E2 30348.417} C_VEL
LIN {X 0,Y 689.46,Z 1117.784,A -85,B 0,C 180,E1 30347.114,E2 30347.114} C_VEL
LIN {X 0,Y 689.017,Z 1132.965,A -85,B 0,C 180,E1 30345.659,E2 30345.659} C_VEL
LIN {X 0,Y 688.652,Z 1147.014,A -85,B 0,C 180,E1 30344.091,E2 30344.091} C_VEL
LIN {X 0,Y 688.385,Z 1159.207,A -85,B 0,C 180,E1 30342.499,E2 30342.499} C_VEL
LIN {X 0,Y 688.182,Z 1169.6,A -85,B 0,C 180,E1 30340.887,E2 30340.887} C_VEL
LIN {X 0,Y 688.052,Z 1178.666,A -85,B 0,C 180,E1 30339.198,E2 30339.198} C_VEL
LIN {X 0,Y 687.97,Z 1186.39,A -85,B 0,C 180,E1 30337.432,E2 30337.432} C_VEL
LIN {X 0,Y 687.922,Z 1192.28,A -85,B 0,C 180,E1 30335.672,E2 30335.672} C_VEL
LIN {X 0,Y 687.915,Z 1196.7,A -85,B 0,C 180,E1 30333.834,E2 30333.834} C_VEL
LIN {X 0,Y 687.917,Z 1199.44,A -85,B 0,C 180,E1 30331.999,E2 30331.999} C_VEL
LIN {X 0,Y 687.907,Z 1200.448,A -85,B 0,C 180,E1 30330.167,E2 30330.167} C_VEL
LIN {X 0,Y 687.907,Z 1199.786,A -85,B 0,C 180,E1 30328.334,E2 30328.334} C_VEL
LIN {X 0,Y 687.911,Z 1197.501,A -85,B 0,C 180,E1 30326.5,E2 30326.5} C_VEL
LIN {X 0,Y 687.926,Z 1193.688,A -85,B 0,C 180,E1 30324.746,E2 30324.746} C_VEL
LIN {X 0,Y 687.949,Z 1188.23,A -85,B 0,C 180,E1 30322.988,E2 30322.988} C_VEL
LIN {X 0,Y 688.027,Z 1181.126,A -85,B 0,C 180,E1 30321.223,E2 30321.223} C_VEL
LIN {X 0,Y 688.144,Z 1172.541,A -85,B 0,C 180,E1 30319.536,E2 30319.536} C_VEL
LIN {X 0,Y 688.316,Z 1162.122,A -85,B 0,C 180,E1 30317.841,E2 30317.841} C_VEL
LIN {X 0,Y 688.576,Z 1150.335,A -85,B 0,C 180,E1 30316.223,E2 30316.223} C_VEL
LIN {X 0,Y 688.912,Z 1137.092,A -85,B 0,C 180,E1 30314.684,E2 30314.684} C_VEL
LIN {X 0,Y 689.323,Z 1122.269,A -85,B 0,C 180,E1 30313.208,E2 30313.208} C_VEL
LIN {X 0,Y 689.818,Z 1106.084,A -85,B 0,C 180,E1 30311.82,E2 30311.82} C_VEL
LIN {X 0,Y 690.372,Z 1088.732,A -85,B 0,C 180,E1 30310.54,E2 30310.54} C_VEL
LIN {X 0,Y 690.934,Z 1070.735,A -85,B 0,C 180,E1 30309.412,E2 30309.412} C_VEL
LIN {X 0,Y 691.55,Z 1051.086,A -85,B 0,C 180,E1 30308.366,E2 30308.366} C_VEL
LIN {X 0,Y 692.111,Z 1031.556,A -85,B 0,C 180,E1 30307.491,E2 30307.491} C_VEL
LIN {X 0,Y 692.648,Z 1011.177,A -85,B 0,C 180,E1 30306.746,E2 30306.746} C_VEL
LIN {X 0,Y 693.109,Z 989.618,A -85,B 0,C 180,E1 30306.123,E2 30306.123} C_VEL
LIN {X 0,Y 693.516,Z 967.693,A -85,B 0,C 180,E1 30305.647,E2 30305.647} C_VEL
LIN {X 0,Y 693.777,Z 945.997,A -85,B 0,C 180,E1 30305.327,E2 30305.327} C_VEL
LIN {X 0,Y 695.286,Z 671.93,A -85,B 0,C 180,E1 30302.292,E2 30302.292} C_VEL
LIN {X 0,Y 695.1,Z 661.203,A -85,B 0,C 180,E1 30302.162,E2 30302.162} C_VEL
LIN {X 0,Y 693.335,Z 650.681,A -85,B 0,C 180,E1 30301.926,E2 30301.926} C_VEL
LIN {X 0,Y 694.428,Z 604.795,A -85,B 0,C 180,E1 30299.112,E2 30299.112} C_VEL
LIN {X 0,Y 695.777,Z 556.234,A -85,B 0,C 180,E1 30296.058,E2 30296.058} C_VEL
LIN {X 0,Y 697.134,Z 510.784,A -85,B 0,C 180,E1 30293.114,E2 30293.114} C_VEL
LIN {X 0,Y 696.69,Z 508.509,A -85,B 0,C 180,E1 30292.932,E2 30292.932} C_VEL
LIN {X 0,Y 688.475,Z 487.704,A -85,B 0,C 180,E1 30290.929,E2 30290.929} C_VEL
LIN {X 0,Y 688.456,Z 487.464,A -85,B 0,C 180,E1 30288.165,E2 30288.165} C_VEL
LIN {X 0,Y 688.428,Z 487.474,A -85,B 0,C 180,E1 30285.219,E2 30285.219} C_VEL
LIN {X 0,Y 688.458,Z 487.458,A -85,B 0,C 180,E1 30282.256,E2 30282.256} C_VEL
LIN {X 0,Y 688.437,Z 487.467,A -85,B 0,C 180,E1 30279.276,E2 30279.276} C_VEL
LIN {X 0,Y 688.456,Z 487.464,A -85,B 0,C 180,E1 30276.29,E2 30276.29} C_VEL
LIN {X 0,Y 688.442,Z 487.465,A -85,B 0,C 180,E1 30273.2,E2 30273.2} C_VEL
LIN {X 0,Y 688.449,Z 487.473,A -85,B 0,C 180,E1 30270.216,E2 30270.216} C_VEL
LIN {X 0,Y 688.443,Z 487.464,A -85,B 0,C 180,E1 30267.039,E2 30267.039} C_VEL
LIN {X 0,Y 688.442,Z 487.477,A -85,B 0,C 180,E1 30264.087,E2 30264.087} C_VEL
LIN {X 0,Y 688.449,Z 487.468,A -85,B 0,C 180,E1 30260.934,E2 30260.934} C_VEL
LIN {X 0,Y 688.431,Z 487.469,A -85,B 0,C 180,E1 30258.021,E2 30258.021} C_VEL
LIN {X 0,Y 688.463,Z 487.46,A -85,B 0,C 180,E1 30254.896,E2 30254.896} C_VEL
LIN {X 0,Y 688.423,Z 487.474,A -85,B 0,C 180,E1 30251.988,E2 30251.988} C_VEL
LIN {X 0,Y 688.461,Z 487.471,A -85,B 0,C 180,E1 30249.024,E2 30249.024} C_VEL
LIN {X 0,Y 688.418,Z 487.467,A -85,B 0,C 180,E1 30246.086,E2 30246.086} C_VEL
LIN {X 0,Y 688.462,Z 487.475,A -85,B 0,C 180,E1 30243.164,E2 30243.164} C_VEL
LIN {X 0,Y 688.43,Z 487.467,A -85,B 0,C 180,E1 30240.166,E2 30240.166} C_VEL
LIN {X 0,Y 688.431,Z 487.476,A -85,B 0,C 180,E1 30237.336,E2 30237.336} C_VEL
LIN {X 0,Y 688.444,Z 487.468,A -85,B 0,C 180,E1 30234.165,E2 30234.165} C_VEL
LIN {X 0,Y 688.42,Z 487.466,A -85,B 0,C 180,E1 30231.312,E2 30231.312} C_VEL
LIN {X 0,Y 688.464,Z 487.463,A -85,B 0,C 180,E1 30228.268,E2 30228.268} C_VEL
LIN {X 0,Y 688.41,Z 487.473,A -85,B 0,C 180,E1 30225.361,E2 30225.361} C_VEL
LIN {X 0,Y 688.465,Z 487.47,A -85,B 0,C 180,E1 30222.504,E2 30222.504} C_VEL
LIN {X 0,Y 688.42,Z 487.466,A -85,B 0,C 180,E1 30219.51,E2 30219.51} C_VEL
LIN {X 0,Y 688.427,Z 487.476,A -85,B 0,C 180,E1 30216.73,E2 30216.73} C_VEL
LIN {X 0,Y 688.445,Z 487.47,A -85,B 0,C 180,E1 30213.613,E2 30213.613} C_VEL
LIN {X 0,Y 688.411,Z 487.471,A -85,B 0,C 180,E1 30210.789,E2 30210.789} C_VEL
LIN {X 0,Y 688.463,Z 487.454,A -85,B 0,C 180,E1 30207.854,E2 30207.854} C_VEL
LIN {X 0,Y 688.41,Z 487.469,A -85,B 0,C 180,E1 30204.99,E2 30204.99} C_VEL
LIN {X 0,Y 688.433,Z 487.468,A -85,B 0,C 180,E1 30202.194,E2 30202.194} C_VEL
LIN {X 0,Y 688.426,Z 487.473,A -85,B 0,C 180,E1 30199.046,E2 30199.046} C_VEL
LIN {X 0,Y 688.41,Z 487.459,A -85,B 0,C 180,E1 30196.261,E2 30196.261} C_VEL
LIN {X 0,Y 688.463,Z 487.462,A -85,B 0,C 180,E1 30193.274,E2 30193.274} C_VEL
LIN {X 0,Y 688.404,Z 487.483,A -85,B 0,C 180,E1 30190.375,E2 30190.375} C_VEL
LIN {X 0,Y 688.505,Z 487.753,A -85,B 0,C 180,E1 30189.371,E2 30189.371} C_VEL
LIN {X 0,Y 697.62,Z 510.239,A -85,B 0,C 180,E1 30187.299,E2 30187.299} C_VEL
LIN {X 0,Y 697.215,Z 528.47,A -85,B 0,C 180,E1 30186.202,E2 30186.202} C_VEL
LIN {X 0,Y 700.182,Z 543.675,A -85,B 0,C 180,E1 30185.834,E2 30185.834} C_VEL
LIN {X 0,Y 698.24,Z 798.539,A -85,B 0,C 180,E1 30182.837,E2 30182.837} C_VEL
LIN {X 0,Y 697.349,Z 919.443,A -85,B 0,C 180,E1 30181.417,E2 30181.417} C_VEL
LIN {X 0,Y 696.828,Z 945.072,A -85,B 0,C 180,E1 30180.966,E2 30180.966} C_VEL
LIN {X 0,Y 696.269,Z 966.82,A -85,B 0,C 180,E1 30180.447,E2 30180.447} C_VEL
LIN {X 0,Y 695.588,Z 991.872,A -85,B 0,C 180,E1 30179.682,E2 30179.682} C_VEL
LIN {X 0,Y 694.878,Z 1012.511,A -85,B 0,C 180,E1 30178.912,E2 30178.912} C_VEL
LIN {X 0,Y 694.05,Z 1035.182,A -85,B 0,C 180,E1 30177.917,E2 30177.917} C_VEL
LIN {X 0,Y 693.229,Z 1055.966,A -85,B 0,C 180,E1 30176.836,E2 30176.836} C_VEL
LIN {X 0,Y 692.398,Z 1076.375,A -85,B 0,C 180,E1 30175.626,E2 30175.626} C_VEL
LIN {X 0,Y 691.566,Z 1096.458,A -85,B 0,C 180,E1 30174.243,E2 30174.243} C_VEL
LIN {X 0,Y 690.816,Z 1115.245,A -85,B 0,C 180,E1 30172.78,E2 30172.78} C_VEL
LIN {X 0,Y 690.135,Z 1132.47,A -85,B 0,C 180,E1 30171.235,E2 30171.235} C_VEL
LIN {X 0,Y 689.56,Z 1148.976,A -85,B 0,C 180,E1 30169.569,E2 30169.569} C_VEL
LIN {X 0,Y 689.063,Z 1163.937,A -85,B 0,C 180,E1 30167.828,E2 30167.828} C_VEL
LIN {X 0,Y 688.663,Z 1178.228,A -85,B 0,C 180,E1 30165.927,E2 30165.927} C_VEL
LIN {X 0,Y 688.376,Z 1189.842,A -85,B 0,C 180,E1 30164.124,E2 30164.124} C_VEL
LIN {X 0,Y 688.165,Z 1200.71,A -85,B 0,C 180,E1 30162.162,E2 30162.162} C_VEL
LIN {X 0,Y 688.037,Z 1209.252,A -85,B 0,C 180,E1 30160.297,E2 30160.297} C_VEL
LIN {X 0,Y 687.975,Z 1216.334,A -85,B 0,C 180,E1 30158.441,E2 30158.441} C_VEL
LIN {X 0,Y 687.929,Z 1222.278,A -85,B 0,C 180,E1 30156.426,E2 30156.426} C_VEL
LIN {X 0,Y 687.915,Z 1226.132,A -85,B 0,C 180,E1 30154.669,E2 30154.669} C_VEL
LIN {X 0,Y 687.887,Z 1229.092,A -85,B 0,C 180,E1 30152.666,E2 30152.666} C_VEL
LIN {X 0,Y 687.885,Z 1230.306,A -85,B 0,C 180,E1 30150.75,E2 30150.75} C_VEL
LIN {X 0,Y 687.899,Z 1230.239,A -85,B 0,C 180,E1 30149.001,E2 30149.001} C_VEL
LIN {X 0,Y 687.886,Z 1228.573,A -85,B 0,C 180,E1 30146.917,E2 30146.917} C_VEL
LIN {X 0,Y 687.903,Z 1225.815,A -85,B 0,C 180,E1 30145.164,E2 30145.164} C_VEL
LIN {X 0,Y 687.936,Z 1221.451,A -85,B 0,C 180,E1 30143.239,E2 30143.239} C_VEL
LIN {X 0,Y 687.966,Z 1215.121,A -85,B 0,C 180,E1 30141.222,E2 30141.222} C_VEL
LIN {X 0,Y 688.058,Z 1208.541,A -85,B 0,C 180,E1 30139.534,E2 30139.534} C_VEL
LIN {X 0,Y 688.201,Z 1198.948,A -85,B 0,C 180,E1 30137.498,E2 30137.498} C_VEL
LIN {X 0,Y 688.395,Z 1188.806,A -85,B 0,C 180,E1 30135.705,E2 30135.705} C_VEL
LIN {X 0,Y 688.706,Z 1176.44,A -85,B 0,C 180,E1 30133.815,E2 30133.815} C_VEL
LIN {X 0,Y 689.088,Z 1163.233,A -85,B 0,C 180,E1 30132.085,E2 30132.085} C_VEL
LIN {X 0,Y 689.59,Z 1148.179,A -85,B 0,C 180,E1 30130.343,E2 30130.343} C_VEL
LIN {X 0,Y 690.169,Z 1131.565,A -85,B 0,C 180,E1 30128.679,E2 30128.679} C_VEL
LIN {X 0,Y 690.876,Z 1113.619,A -85,B 0,C 180,E1 30127.089,E2 30127.089} C_VEL
LIN {X 0,Y 691.588,Z 1095.849,A -85,B 0,C 180,E1 30125.713,E2 30125.713} C_VEL
LIN {X 0,Y 692.427,Z 1075.642,A -85,B 0,C 180,E1 30124.329,E2 30124.329} C_VEL
LIN {X 0,Y 693.227,Z 1055.961,A -85,B 0,C 180,E1 30123.163,E2 30123.163} C_VEL
LIN {X 0,Y 694.091,Z 1034.169,A -85,B 0,C 180,E1 30122.033,E2 30122.033} C_VEL
LIN {X 0,Y 694.878,Z 1012.513,A -85,B 0,C 180,E1 30121.088,E2 30121.088} C_VEL
LIN {X 0,Y 695.638,Z 990.587,A -85,B 0,C 180,E1 30120.272,E2 30120.272} C_VEL
LIN {X 0,Y 696.283,Z 966.155,A -85,B 0,C 180,E1 30119.536,E2 30119.536} C_VEL
LIN {X 0,Y 696.855,Z 944.293,A -85,B 0,C 180,E1 30119.017,E2 30119.017} C_VEL
LIN {X 0,Y 697.353,Z 918.855,A -85,B 0,C 180,E1 30118.575,E2 30118.575} C_VEL
LIN {X 0,Y 699.192,Z 666.467,A -85,B 0,C 180,E1 30115.619,E2 30115.619} C_VEL
LIN {X 0,Y 700,Z 541.719,A -85,B 0,C 180,E1 30114.131,E2 30114.131} C_VEL
LIN {X 0,Y 697.152,Z 527.956,A -85,B 0,C 180,E1 30113.78,E2 30113.78} C_VEL
LIN {X 0,Y 697.499,Z 509.917,A -85,B 0,C 180,E1 30112.673,E2 30112.673} C_VEL
LIN {X 0,Y 688.505,Z 487.753,A -85,B 0,C 180,E1 30110.629,E2 30110.629} C_VEL
LIN {X 0,Y 688.405,Z 487.482,A -85,B 0,C 180,E1 30109.516,E2 30109.516} C_VEL
LIN {X 0,Y 688.465,Z 487.464,A -85,B 0,C 180,E1 30106.567,E2 30106.567} C_VEL
LIN {X 0,Y 688.405,Z 487.46,A -85,B 0,C 180,E1 30103.624,E2 30103.624} C_VEL
LIN {X 0,Y 688.442,Z 487.472,A -85,B 0,C 180,E1 30100.812,E2 30100.812} C_VEL
LIN {X 0,Y 688.423,Z 487.473,A -85,B 0,C 180,E1 30097.669,E2 30097.669} C_VEL
LIN {X 0,Y 688.422,Z 487.467,A -85,B 0,C 180,E1 30094.855,E2 30094.855} C_VEL
LIN {X 0,Y 688.448,Z 487.466,A -85,B 0,C 180,E1 30091.72,E2 30091.72} C_VEL
LIN {X 0,Y 688.41,Z 487.469,A -85,B 0,C 180,E1 30088.926,E2 30088.926} C_VEL
LIN {X 0,Y 688.464,Z 487.472,A -85,B 0,C 180,E1 30085.977,E2 30085.977} C_VEL
LIN {X 0,Y 688.414,Z 487.474,A -85,B 0,C 180,E1 30082.999,E2 30082.999} C_VEL
LIN {X 0,Y 688.454,Z 487.464,A -85,B 0,C 180,E1 30080.134,E2 30080.134} C_VEL
LIN {X 0,Y 688.43,Z 487.471,A -85,B 0,C 180,E1 30077.061,E2 30077.061} C_VEL
LIN {X 0,Y 688.43,Z 487.47,A -85,B 0,C 180,E1 30074.209,E2 30074.209} C_VEL
LIN {X 0,Y 688.449,Z 487.478,A -85,B 0,C 180,E1 30071.053,E2 30071.053} C_VEL
LIN {X 0,Y 688.422,Z 487.462,A -85,B 0,C 180,E1 30068.183,E2 30068.183} C_VEL
LIN {X 0,Y 688.462,Z 487.475,A -85,B 0,C 180,E1 30065.166,E2 30065.166} C_VEL
LIN {X 0,Y 688.419,Z 487.471,A -85,B 0,C 180,E1 30062.225,E2 30062.225} C_VEL
LIN {X 0,Y 688.462,Z 487.465,A -85,B 0,C 180,E1 30059.334,E2 30059.334} C_VEL
LIN {X 0,Y 688.429,Z 487.474,A -85,B 0,C 180,E1 30056.336,E2 30056.336} C_VEL
LIN {X 0,Y 688.454,Z 487.462,A -85,B 0,C 180,E1 30053.407,E2 30053.407} C_VEL
LIN {X 0,Y 688.44,Z 487.468,A -85,B 0,C 180,E1 30050.301,E2 30050.301} C_VEL
LIN {X 0,Y 688.446,Z 487.468,A -85,B 0,C 180,E1 30047.331,E2 30047.331} C_VEL
LIN {X 0,Y 688.448,Z 487.477,A -85,B 0,C 180,E1 30044.154,E2 30044.154} C_VEL
LIN {X 0,Y 688.443,Z 487.462,A -85,B 0,C 180,E1 30041.19,E2 30041.19} C_VEL
LIN {X 0,Y 688.459,Z 487.472,A -85,B 0,C 180,E1 30038.083,E2 30038.083} C_VEL
LIN {X 0,Y 688.437,Z 487.469,A -85,B 0,C 180,E1 30035.09,E2 30035.09} C_VEL
LIN {X 0,Y 688.455,Z 487.468,A -85,B 0,C 180,E1 30032.312,E2 30032.312} C_VEL
LIN {X 0,Y 687.467,Z 487.6,A -85,B 0,C 180,E1 30031.671,E2 30031.671} C_VEL
LIN {X 0,Y 681.04,Z 488.4,A -85,B 0,C 180,E1 30029.874,E2 30029.874} C_VEL
LIN {X 0,Y 680.493,Z 488.462,A -85,B 0,C 180,E1 30029.407,E2 30029.407} C_VEL
LIN {X 0,Y 680.521,Z 488.453,A -85,B 0,C 180,E1 30026.415,E2 30026.415} C_VEL
LIN {X 0,Y 680.497,Z 488.448,A -85,B 0,C 180,E1 30023.344,E2 30023.344} C_VEL
LIN {X 0,Y 680.525,Z 488.454,A -85,B 0,C 180,E1 30020.343,E2 30020.343} C_VEL
LIN {X 0,Y 680.504,Z 488.442,A -85,B 0,C 180,E1 30017.247,E2 30017.247} C_VEL
LIN {X 0,Y 680.524,Z 488.458,A -85,B 0,C 180,E1 30014.191,E2 30014.191} C_VEL
LIN {X 0,Y 680.509,Z 488.467,A -85,B 0,C 180,E1 30011.054,E2 30011.054} C_VEL
LIN {X 0,Y 680.549,Z 488.678,A -85,B 0,C 180,E1 30009.451,E2 30009.451} C_VEL
LIN {X 0,Y 690.116,Z 512.808,A -85,B 0,C 180,E1 30007.098,E2 30007.098} C_VEL
LIN {X 0,Y 689.039,Z 547.484,A -85,B 0,C 180,E1 30004.815,E2 30004.815} C_VEL
LIN {X 0,Y 687.636,Z 593.651,A -85,B 0,C 180,E1 30001.858,E2 30001.858} C_VEL
LIN {X 0,Y 686.288,Z 640.639,A -85,B 0,C 180,E1 29998.927,E2 29998.927} C_VEL
LIN {X 0,Y 686.14,Z 650.902,A -85,B 0,C 180,E1 29998.323,E2 29998.323} C_VEL
LIN {X 0,Y 688.407,Z 665.02,A -85,B 0,C 180,E1 29998.03,E2 29998.03} C_VEL
LIN {X 0,Y 686.736,Z 908.775,A -85,B 0,C 180,E1 29995.277,E2 29995.277} C_VEL
LIN {X 0,Y 686.378,Z 958.122,A -85,B 0,C 180,E1 29994.702,E2 29994.702} C_VEL
LIN {X 0,Y 685.975,Z 979.862,A -85,B 0,C 180,E1 29994.293,E2 29994.293} C_VEL
LIN {X 0,Y 685.495,Z 1001.238,A -85,B 0,C 180,E1 29993.739,E2 29993.739} C_VEL
LIN {X 0,Y 684.966,Z 1021.391,A -85,B 0,C 180,E1 29993.075,E2 29993.075} C_VEL
LIN {X 0,Y 684.324,Z 1041.761,A -85,B 0,C 180,E1 29992.236,E2 29992.236} C_VEL
LIN {X 0,Y 683.661,Z 1061.319,A -85,B 0,C 180,E1 29991.266,E2 29991.266} C_VEL
LIN {X 0,Y 682.999,Z 1080.092,A -85,B 0,C 180,E1 29990.167,E2 29990.167} C_VEL
LIN {X 0,Y 682.371,Z 1097.816,A -85,B 0,C 180,E1 29988.945,E2 29988.945} C_VEL
LIN {X 0,Y 681.79,Z 1114.166,A -85,B 0,C 180,E1 29987.628,E2 29987.628} C_VEL
LIN {X 0,Y 681.275,Z 1129.587,A -85,B 0,C 180,E1 29986.191,E2 29986.191} C_VEL
LIN {X 0,Y 680.848,Z 1143.979,A -85,B 0,C 180,E1 29984.631,E2 29984.631} C_VEL
LIN {X 0,Y 680.512,Z 1156.759,A -85,B 0,C 180,E1 29982.991,E2 29982.991} C_VEL
LIN {X 0,Y 680.264,Z 1167.544,A -85,B 0,C 180,E1 29981.359,E2 29981.359} C_VEL
LIN {X 0,Y 680.102,Z 1177.045,A -85,B 0,C 180,E1 29979.648,E2 29979.648} C_VEL
LIN {X 0,Y 679.998,Z 1184.691,A -85,B 0,C 180,E1 29977.945,E2 29977.945} C_VEL
LIN {X 0,Y 679.936,Z 1191.268,A -85,B 0,C 180,E1 29976.078,E2 29976.078} C_VEL
LIN {X 0,Y 679.926,Z 1195.899,A -85,B 0,C 180,E1 29974.301,E2 29974.301} C_VEL
LIN {X 0,Y 679.914,Z 1198.84,A -85,B 0,C 180,E1 29972.529,E2 29972.529} C_VEL
LIN {X 0,Y 679.905,Z 1200.337,A -85,B 0,C 180,E1 29970.59,E2 29970.59} C_VEL
LIN {X 0,Y 679.905,Z 1200.185,A -85,B 0,C 180,E1 29968.82,E2 29968.82} C_VEL
LIN {X 0,Y 679.911,Z 1198.283,A -85,B 0,C 180,E1 29966.965,E2 29966.965} C_VEL
LIN {X 0,Y 679.915,Z 1194.717,A -85,B 0,C 180,E1 29965.107,E2 29965.107} C_VEL
LIN {X 0,Y 679.943,Z 1189.74,A -85,B 0,C 180,E1 29963.329,E2 29963.329} C_VEL
LIN {X 0,Y 680.027,Z 1182.945,A -85,B 0,C 180,E1 29961.545,E2 29961.545} C_VEL
LIN {X 0,Y 680.14,Z 1174.378,A -85,B 0,C 180,E1 29959.754,E2 29959.754} C_VEL
LIN {X 0,Y 680.325,Z 1164.413,A -85,B 0,C 180,E1 29958.04,E2 29958.04} C_VEL
LIN {X 0,Y 680.596,Z 1152.967,A -85,B 0,C 180,E1 29956.405,E2 29956.405} C_VEL
LIN {X 0,Y 680.957,Z 1140.18,A -85,B 0,C 180,E1 29954.849,E2 29954.849} C_VEL
LIN {X 0,Y 681.393,Z 1126.128,A -85,B 0,C 180,E1 29953.373,E2 29953.373} C_VEL
LIN {X 0,Y 681.923,Z 1110.275,A -85,B 0,C 180,E1 29951.947,E2 29951.947} C_VEL
LIN {X 0,Y 682.515,Z 1093.359,A -85,B 0,C 180,E1 29950.643,E2 29950.643} C_VEL
LIN {X 0,Y 683.205,Z 1074.355,A -85,B 0,C 180,E1 29949.389,E2 29949.389} C_VEL
LIN {X 0,Y 683.877,Z 1055.372,A -85,B 0,C 180,E1 29948.326,E2 29948.326} C_VEL
LIN {X 0,Y 684.52,Z 1035.718,A -85,B 0,C 180,E1 29947.409,E2 29947.409} C_VEL
LIN {X 0,Y 685.127,Z 1015.018,A -85,B 0,C 180,E1 29946.612,E2 29946.612} C_VEL
LIN {X 0,Y 685.687,Z 993.84,A -85,B 0,C 180,E1 29945.96,E2 29945.96} C_VEL
LIN {X 0,Y 686.127,Z 972.619,A -85,B 0,C 180,E1 29945.464,E2 29945.464} C_VEL
LIN {X 0,Y 686.442,Z 950.752,A -85,B 0,C 180,E1 29945.109,E2 29945.109} C_VEL
LIN {X 0,Y 688.315,Z 676.232,A -85,B 0,C 180,E1 29942.009,E2 29942.009} C_VEL
LIN {X 0,Y 688.202,Z 662.586,A -85,B 0,C 180,E1 29941.84,E2 29941.84} C_VEL
LIN {X 0,Y 686.068,Z 650.2,A -85,B 0,C 180,E1 29941.563,E2 29941.563} C_VEL
LIN {X 0,Y 687.247,Z 605.66,A -85,B 0,C 180,E1 29938.806,E2 29938.806} C_VEL
LIN {X 0,Y 688.761,Z 557.104,A -85,B 0,C 180,E1 29935.719,E2 29935.719} C_VEL
LIN {X 0,Y 690.21,Z 513.094,A -85,B 0,C 180,E1 29932.838,E2 29932.838} C_VEL
LIN {X 0,Y 681.606,Z 491.603,A -85,B 0,C 180,E1 29930.765,E2 29930.765} C_VEL
LIN {X 0,Y 680.543,Z 488.633,A -85,B 0,C 180,E1 29930.439,E2 29930.439} C_VEL
LIN {X 0,Y 680.496,Z 488.442,A -85,B 0,C 180,E1 29927.477,E2 29927.477} C_VEL
LIN {X 0,Y 680.521,Z 488.46,A -85,B 0,C 180,E1 29924.496,E2 29924.496} C_VEL
LIN {X 0,Y 680.498,Z 488.456,A -85,B 0,C 180,E1 29921.339,E2 29921.339} C_VEL
LIN {X 0,Y 680.512,Z 488.443,A -85,B 0,C 180,E1 29918.428,E2 29918.428} C_VEL
LIN {X 0,Y 680.506,Z 488.459,A -85,B 0,C 180,E1 29915.272,E2 29915.272} C_VEL
LIN {X 0,Y 680.514,Z 488.463,A -85,B 0,C 180,E1 29912.233,E2 29912.233} C_VEL
LIN {X 0,Y 680.505,Z 488.457,A -85,B 0,C 180,E1 29909.101,E2 29909.101} C_VEL
LIN {X 0,Y 680.505,Z 488.459,A -85,B 0,C 180,E1 29906.138,E2 29906.138} C_VEL
LIN {X 0,Y 680.512,Z 488.449,A -85,B 0,C 180,E1 29903.007,E2 29903.007} C_VEL
LIN {X 0,Y 680.498,Z 488.465,A -85,B 0,C 180,E1 29900.021,E2 29900.021} C_VEL
LIN {X 0,Y 680.518,Z 488.456,A -85,B 0,C 180,E1 29896.913,E2 29896.913} C_VEL
LIN {X 0,Y 680.487,Z 488.457,A -85,B 0,C 180,E1 29893.944,E2 29893.944} C_VEL
LIN {X 0,Y 680.522,Z 488.449,A -85,B 0,C 180,E1 29890.926,E2 29890.926} C_VEL
LIN {X 0,Y 680.481,Z 488.462,A -85,B 0,C 180,E1 29887.973,E2 29887.973} C_VEL
LIN {X 0,Y 680.522,Z 488.461,A -85,B 0,C 180,E1 29885.029,E2 29885.029} C_VEL
LIN {X 0,Y 680.479,Z 488.458,A -85,B 0,C 180,E1 29882.021,E2 29882.021} C_VEL
LIN {X 0,Y 680.525,Z 488.466,A -85,B 0,C 180,E1 29879.074,E2 29879.074} C_VEL
LIN {X 0,Y 680.488,Z 488.453,A -85,B 0,C 180,E1 29876.04,E2 29876.04} C_VEL
LIN {X 0,Y 680.497,Z 488.466,A -85,B 0,C 180,E1 29873.165,E2 29873.165} C_VEL
LIN {X 0,Y 680.502,Z 488.458,A -85,B 0,C 180,E1 29870.015,E2 29870.015} C_VEL
LIN {X 0,Y 680.482,Z 488.458,A -85,B 0,C 180,E1 29867.181,E2 29867.181} C_VEL
LIN {X 0,Y 680.526,Z 488.453,A -85,B 0,C 180,E1 29864.14,E2 29864.14} C_VEL
LIN {X 0,Y 680.473,Z 488.462,A -85,B 0,C 180,E1 29861.228,E2 29861.228} C_VEL
LIN {X 0,Y 680.526,Z 488.461,A -85,B 0,C 180,E1 29858.268,E2 29858.268} C_VEL
LIN {X 0,Y 680.477,Z 488.454,A -85,B 0,C 180,E1 29855.335,E2 29855.335} C_VEL
LIN {X 0,Y 680.496,Z 488.467,A -85,B 0,C 180,E1 29852.524,E2 29852.524} C_VEL
LIN {X 0,Y 680.489,Z 488.459,A -85,B 0,C 180,E1 29849.345,E2 29849.345} C_VEL
LIN {X 0,Y 680.476,Z 488.441,A -85,B 0,C 180,E1 29846.562,E2 29846.562} C_VEL
LIN {X 0,Y 680.519,Z 488.459,A -85,B 0,C 180,E1 29843.482,E2 29843.482} C_VEL
LIN {X 0,Y 680.464,Z 488.44,A -85,B 0,C 180,E1 29840.595,E2 29840.595} C_VEL
LIN {X 0,Y 680.525,Z 488.454,A -85,B 0,C 180,E1 29837.706,E2 29837.706} C_VEL
LIN {X 0,Y 680.472,Z 488.464,A -85,B 0,C 180,E1 29834.734,E2 29834.734} C_VEL
LIN {X 0,Y 680.484,Z 488.441,A -85,B 0,C 180,E1 29831.955,E2 29831.955} C_VEL
LIN {X 0,Y 680.518,Z 488.667,A -85,B 0,C 180,E1 29829.87,E2 29829.87} C_VEL
LIN {X 0,Y 683.122,Z 495.138,A -85,B 0,C 180,E1 29829.22,E2 29829.22} C_VEL
LIN {X 0,Y 690.715,Z 513.749,A -85,B 0,C 180,E1 29827.505,E2 29827.505} C_VEL
LIN {X 0,Y 690.335,Z 529.213,A -85,B 0,C 180,E1 29826.568,E2 29826.568} C_VEL
LIN {X 0,Y 693.622,Z 545.187,A -85,B 0,C 180,E1 29826.197,E2 29826.197} C_VEL
LIN {X 0,Y 691.512,Z 799.048,A -85,B 0,C 180,E1 29823.191,E2 29823.191} C_VEL
LIN {X 0,Y 690.512,Z 919.514,A -85,B 0,C 180,E1 29821.763,E2 29821.763} C_VEL
LIN {X 0,Y 689.946,Z 945.07,A -85,B 0,C 180,E1 29821.31,E2 29821.31} C_VEL
LIN {X 0,Y 689.322,Z 966.709,A -85,B 0,C 180,E1 29820.79,E2 29820.79} C_VEL
LIN {X 0,Y 688.554,Z 991.869,A -85,B 0,C 180,E1 29820.017,E2 29820.017} C_VEL
LIN {X 0,Y 687.77,Z 1012.507,A -85,B 0,C 180,E1 29819.24,E2 29819.24} C_VEL
LIN {X 0,Y 686.833,Z 1035.178,A -85,B 0,C 180,E1 29818.237,E2 29818.237} C_VEL
LIN {X 0,Y 685.914,Z 1055.962,A -85,B 0,C 180,E1 29817.146,E2 29817.146} C_VEL
LIN {X 0,Y 684.995,Z 1076.377,A -85,B 0,C 180,E1 29815.923,E2 29815.923} C_VEL
LIN {X 0,Y 684.045,Z 1096.456,A -85,B 0,C 180,E1 29814.527,E2 29814.527} C_VEL
LIN {X 0,Y 683.211,Z 1115.26,A -85,B 0,C 180,E1 29813.046,E2 29813.046} C_VEL
LIN {X 0,Y 682.439,Z 1132.468,A -85,B 0,C 180,E1 29811.486,E2 29811.486} C_VEL
LIN {X 0,Y 681.789,Z 1148.978,A -85,B 0,C 180,E1 29809.802,E2 29809.802} C_VEL
LIN {X 0,Y 681.23,Z 1163.935,A -85,B 0,C 180,E1 29808.04,E2 29808.04} C_VEL
LIN {X 0,Y 680.768,Z 1178.23,A -85,B 0,C 180,E1 29806.116,E2 29806.116} C_VEL
LIN {X 0,Y 680.441,Z 1189.841,A -85,B 0,C 180,E1 29804.292,E2 29804.292} C_VEL
LIN {X 0,Y 680.205,Z 1200.711,A -85,B 0,C 180,E1 29802.306,E2 29802.306} C_VEL
LIN {X 0,Y 680.062,Z 1209.408,A -85,B 0,C 180,E1 29800.381,E2 29800.381} C_VEL
LIN {X 0,Y 679.987,Z 1216.936,A -85,B 0,C 180,E1 29798.37,E2 29798.37} C_VEL
LIN {X 0,Y 679.932,Z 1222.484,A -85,B 0,C 180,E1 29796.417,E2 29796.417} C_VEL
LIN {X 0,Y 679.916,Z 1226.291,A -85,B 0,C 180,E1 29794.639,E2 29794.639} C_VEL
LIN {X 0,Y 679.895,Z 1229.227,A -85,B 0,C 180,E1 29792.529,E2 29792.529} C_VEL
LIN {X 0,Y 679.883,Z 1230.328,A -85,B 0,C 180,E1 29790.674,E2 29790.674} C_VEL
LIN {X 0,Y 679.911,Z 1230.193,A -85,B 0,C 180,E1 29788.82,E2 29788.82} C_VEL
LIN {X 0,Y 679.899,Z 1228.349,A -85,B 0,C 180,E1 29786.712,E2 29786.712} C_VEL
LIN {X 0,Y 679.893,Z 1225.497,A -85,B 0,C 180,E1 29784.938,E2 29784.938} C_VEL
LIN {X 0,Y 679.942,Z 1220.762,A -85,B 0,C 180,E1 29782.905,E2 29782.905} C_VEL
LIN {X 0,Y 679.983,Z 1214.818,A -85,B 0,C 180,E1 29781.033,E2 29781.033} C_VEL
LIN {X 0,Y 680.078,Z 1207.831,A -85,B 0,C 180,E1 29779.239,E2 29779.239} C_VEL
LIN {X 0,Y 680.267,Z 1198.03,A -85,B 0,C 180,E1 29777.177,E2 29777.177} C_VEL
LIN {X 0,Y 680.481,Z 1188.288,A -85,B 0,C 180,E1 29775.448,E2 29775.448} C_VEL
LIN {X 0,Y 680.85,Z 1175.168,A -85,B 0,C 180,E1 29773.447,E2 29773.447} C_VEL
LIN {X 0,Y 681.289,Z 1162.066,A -85,B 0,C 180,E1 29771.726,E2 29771.726} C_VEL
LIN {X 0,Y 681.914,Z 1145.643,A -85,B 0,C 180,E1 29769.845,E2 29769.845} C_VEL
LIN {X 0,Y 682.519,Z 1130.614,A -85,B 0,C 180,E1 29768.336,E2 29768.336} C_VEL
LIN {X 0,Y 683.397,Z 1110.857,A -85,B 0,C 180,E1 29766.595,E2 29766.595} C_VEL
LIN {X 0,Y 684.205,Z 1092.804,A -85,B 0,C 180,E1 29765.203,E2 29765.203} C_VEL
LIN {X 0,Y 685.183,Z 1072.011,A -85,B 0,C 180,E1 29763.805,E2 29763.805} C_VEL
LIN {X 0,Y 686.047,Z 1052.712,A -85,B 0,C 180,E1 29762.672,E2 29762.672} C_VEL
LIN {X 0,Y 687.088,Z 1029.304,A -85,B 0,C 180,E1 29761.49,E2 29761.49} C_VEL
LIN {X 0,Y 687.863,Z 1010.249,A -85,B 0,C 180,E1 29760.669,E2 29760.669} C_VEL
LIN {X 0,Y 688.719,Z 987.221,A -85,B 0,C 180,E1 29759.823,E2 29759.823} C_VEL
LIN {X 0,Y 689.403,Z 964.355,A -85,B 0,C 180,E1 29759.149,E2 29759.149} C_VEL
LIN {X 0,Y 690.1,Z 940.809,A -85,B 0,C 180,E1 29758.599,E2 29758.599} C_VEL
LIN {X 0,Y 690.539,Z 916.477,A -85,B 0,C 180,E1 29758.195,E2 29758.195} C_VEL
LIN {X 0,Y 692.598,Z 664.855,A -85,B 0,C 180,E1 29755.225,E2 29755.225} C_VEL
LIN {X 0,Y 693.449,Z 543.42,A -85,B 0,C 180,E1 29753.773,E2 29753.773} C_VEL
LIN {X 0,Y 690.263,Z 528.637,A -85,B 0,C 180,E1 29753.411,E2 29753.411} C_VEL
LIN {X 0,Y 690.62,Z 513.382,A -85,B 0,C 180,E1 29752.466,E2 29752.466} C_VEL
LIN {X 0,Y 681.361,Z 491.159,A -85,B 0,C 180,E1 29750.393,E2 29750.393} C_VEL
LIN {X 0,Y 680.518,Z 488.667,A -85,B 0,C 180,E1 29750.13,E2 29750.13} C_VEL
LIN {X 0,Y 680.464,Z 488.446,A -85,B 0,C 180,E1 29747.475,E2 29747.475} C_VEL
LIN {X 0,Y 680.524,Z 488.445,A -85,B 0,C 180,E1 29744.555,E2 29744.555} C_VEL
LIN {X 0,Y 680.471,Z 488.467,A -85,B 0,C 180,E1 29741.591,E2 29741.591} C_VEL
LIN {X 0,Y 680.501,Z 488.435,A -85,B 0,C 180,E1 29738.751,E2 29738.751} C_VEL
LIN {X 0,Y 680.49,Z 488.462,A -85,B 0,C 180,E1 29735.656,E2 29735.656} C_VEL
LIN {X 0,Y 680.48,Z 488.44,A -85,B 0,C 180,E1 29732.811,E2 29732.811} C_VEL
LIN {X 0,Y 680.515,Z 488.463,A -85,B 0,C 180,E1 29729.68,E2 29729.68} C_VEL
LIN {X 0,Y 680.475,Z 488.462,A -85,B 0,C 180,E1 29726.815,E2 29726.815} C_VEL
LIN {X 0,Y 680.524,Z 488.456,A -85,B 0,C 180,E1 29723.832,E2 29723.832} C_VEL
LIN {X 0,Y 680.476,Z 488.459,A -85,B 0,C 180,E1 29720.92,E2 29720.92} C_VEL
LIN {X 0,Y 680.516,Z 488.457,A -85,B 0,C 180,E1 29718.061,E2 29718.061} C_VEL
LIN {X 0,Y 680.491,Z 488.465,A -85,B 0,C 180,E1 29714.988,E2 29714.988} C_VEL
LIN {X 0,Y 680.493,Z 488.452,A -85,B 0,C 180,E1 29712.129,E2 29712.129} C_VEL
LIN {X 0,Y 680.507,Z 488.457,A -85,B 0,C 180,E1 29708.96,E2 29708.96} C_VEL
LIN {X 0,Y 680.488,Z 488.458,A -85,B 0,C 180,E1 29706.073,E2 29706.073} C_VEL
LIN {X 0,Y 680.522,Z 488.455,A -85,B 0,C 180,E1 29703.032,E2 29703.032} C_VEL
LIN {X 0,Y 680.481,Z 488.457,A -85,B 0,C 180,E1 29700.084,E2 29700.084} C_VEL
LIN {X 0,Y 680.52,Z 488.457,A -85,B 0,C 180,E1 29697.136,E2 29697.136} C_VEL
LIN {X 0,Y 680.486,Z 488.458,A -85,B 0,C 180,E1 29694.181,E2 29694.181} C_VEL
LIN {X 0,Y 680.525,Z 488.456,A -85,B 0,C 180,E1 29691.21,E2 29691.21} C_VEL
LIN {X 0,Y 680.494,Z 488.465,A -85,B 0,C 180,E1 29688.114,E2 29688.114} C_VEL
LIN {X 0,Y 680.525,Z 488.448,A -85,B 0,C 180,E1 29685.1,E2 29685.1} C_VEL
LIN {X 0,Y 680.503,Z 488.459,A -85,B 0,C 180,E1 29682.027,E2 29682.027} C_VEL
LIN {X 0,Y 680.52,Z 488.456,A -85,B 0,C 180,E1 29678.991,E2 29678.991} C_VEL
LIN {X 0,Y 680.506,Z 488.466,A -85,B 0,C 180,E1 29675.843,E2 29675.843} C_VEL
LIN {X 0,Y 680.518,Z 488.451,A -85,B 0,C 180,E1 29672.809,E2 29672.809} C_VEL
LIN {X 0,Y 680.504,Z 488.461,A -85,B 0,C 180,E1 29669.638,E2 29669.638} C_VEL
LIN {X 0,Y 680.493,Z 488.462,A -85,B 0,C 180,E1 29669.407,E2 29669.407} C_VEL
LIN {X 0,Y 679.494,Z 488.587,A -85,B 0,C 180,E1 29668.759,E2 29668.759} C_VEL
LIN {X 0,Y 673.11,Z 489.377,A -85,B 0,C 180,E1 29666.941,E2 29666.941} C_VEL
LIN {X 0,Y 672.583,Z 489.442,A -85,B 0,C 180,E1 29666.468,E2 29666.468} C_VEL
LIN {X 0,Y 672.562,Z 489.436,A -85,B 0,C 180,E1 29663.397,E2 29663.397} C_VEL
LIN {X 0,Y 672.586,Z 489.443,A -85,B 0,C 180,E1 29660.358,E2 29660.358} C_VEL
LIN {X 0,Y 672.566,Z 489.428,A -85,B 0,C 180,E1 29657.256,E2 29657.256} C_VEL
LIN {X 0,Y 672.585,Z 489.447,A -85,B 0,C 180,E1 29654.203,E2 29654.203} C_VEL
LIN {X 0,Y 672.573,Z 489.457,A -85,B 0,C 180,E1 29651.078,E2 29651.078} C_VEL
LIN {X 0,Y 672.621,Z 489.73,A -85,B 0,C 180,E1 29649.93,E2 29649.93} C_VEL
LIN {X 0,Y 682.217,Z 513.726,A -85,B 0,C 180,E1 29647.541,E2 29647.541} C_VEL
LIN {X 0,Y 683.287,Z 516.999,A -85,B 0,C 180,E1 29647.244,E2 29647.244} C_VEL
LIN {X 0,Y 681.583,Z 562.623,A -85,B 0,C 180,E1 29644.234,E2 29644.234} C_VEL
LIN {X 0,Y 680.014,Z 608.869,A -85,B 0,C 180,E1 29641.267,E2 29641.267} C_VEL
LIN {X 0,Y 678.833,Z 649.588,A -85,B 0,C 180,E1 29638.726,E2 29638.726} C_VEL
LIN {X 0,Y 681.618,Z 666.363,A -85,B 0,C 180,E1 29638.373,E2 29638.373} C_VEL
LIN {X 0,Y 679.451,Z 918.024,A -85,B 0,C 180,E1 29635.463,E2 29635.463} C_VEL
LIN {X 0,Y 679.089,Z 958.804,A -85,B 0,C 180,E1 29634.973,E2 29634.973} C_VEL
LIN {X 0,Y 678.656,Z 980.356,A -85,B 0,C 180,E1 29634.562,E2 29634.562} C_VEL
LIN {X 0,Y 678.112,Z 1002.064,A -85,B 0,C 180,E1 29633.988,E2 29633.988} C_VEL
LIN {X 0,Y 677.504,Z 1022.532,A -85,B 0,C 180,E1 29633.298,E2 29633.298} C_VEL
LIN {X 0,Y 676.82,Z 1042.419,A -85,B 0,C 180,E1 29632.466,E2 29632.466} C_VEL
LIN {X 0,Y 676.072,Z 1062.136,A -85,B 0,C 180,E1 29631.471,E2 29631.471} C_VEL
LIN {X 0,Y 675.34,Z 1080.765,A -85,B 0,C 180,E1 29630.36,E2 29630.36} C_VEL
LIN {X 0,Y 674.647,Z 1098.515,A -85,B 0,C 180,E1 29629.119,E2 29629.119} C_VEL
LIN {X 0,Y 674.001,Z 1114.678,A -85,B 0,C 180,E1 29627.794,E2 29627.794} C_VEL
LIN {X 0,Y 673.415,Z 1130.438,A -85,B 0,C 180,E1 29626.297,E2 29626.297} C_VEL
LIN {X 0,Y 672.971,Z 1143.984,A -85,B 0,C 180,E1 29624.806,E2 29624.806} C_VEL
LIN {X 0,Y 672.591,Z 1156.761,A -85,B 0,C 180,E1 29623.147,E2 29623.147} C_VEL
LIN {X 0,Y 672.3,Z 1168.061,A -85,B 0,C 180,E1 29621.408,E2 29621.408} C_VEL
LIN {X 0,Y 672.119,Z 1177.454,A -85,B 0,C 180,E1 29619.677,E2 29619.677} C_VEL
LIN {X 0,Y 672.006,Z 1185.047,A -85,B 0,C 180,E1 29617.954,E2 29617.954} C_VEL
LIN {X 0,Y 671.943,Z 1191.27,A -85,B 0,C 180,E1 29616.15,E2 29616.15} C_VEL
LIN {X 0,Y 671.926,Z 1195.899,A -85,B 0,C 180,E1 29614.352,E2 29614.352} C_VEL
LIN {X 0,Y 671.914,Z 1198.841,A -85,B 0,C 180,E1 29612.559,E2 29612.559} C_VEL
LIN {X 0,Y 671.905,Z 1200.336,A -85,B 0,C 180,E1 29610.597,E2 29610.597} C_VEL
LIN {X 0,Y 671.905,Z 1200.185,A -85,B 0,C 180,E1 29608.806,E2 29608.806} C_VEL
LIN {X 0,Y 671.911,Z 1198.282,A -85,B 0,C 180,E1 29606.929,E2 29606.929} C_VEL
LIN {X 0,Y 671.917,Z 1194.717,A -85,B 0,C 180,E1 29605.049,E2 29605.049} C_VEL
LIN {X 0,Y 671.948,Z 1189.739,A -85,B 0,C 180,E1 29603.249,E2 29603.249} C_VEL
LIN {X 0,Y 672.038,Z 1182.943,A -85,B 0,C 180,E1 29601.444,E2 29601.444} C_VEL
LIN {X 0,Y 672.173,Z 1174.375,A -85,B 0,C 180,E1 29599.631,E2 29599.631} C_VEL
LIN {X 0,Y 672.382,Z 1164.408,A -85,B 0,C 180,E1 29597.897,E2 29597.897} C_VEL
LIN {X 0,Y 672.685,Z 1152.964,A -85,B 0,C 180,E1 29596.242,E2 29596.242} C_VEL
LIN {X 0,Y 673.09,Z 1140.174,A -85,B 0,C 180,E1 29594.668,E2 29594.668} C_VEL
LIN {X 0,Y 673.583,Z 1126.122,A -85,B 0,C 180,E1 29593.175,E2 29593.175} C_VEL
LIN {X 0,Y 674.162,Z 1110.628,A -85,B 0,C 180,E1 29591.764,E2 29591.764} C_VEL
LIN {X 0,Y 674.816,Z 1093.662,A -85,B 0,C 180,E1 29590.436,E2 29590.436} C_VEL
LIN {X 0,Y 675.569,Z 1075.125,A -85,B 0,C 180,E1 29589.194,E2 29589.194} C_VEL
LIN {X 0,Y 676.329,Z 1055.946,A -85,B 0,C 180,E1 29588.102,E2 29588.102} C_VEL
LIN {X 0,Y 677.022,Z 1036.607,A -85,B 0,C 180,E1 29587.186,E2 29587.186} C_VEL
LIN {X 0,Y 677.694,Z 1016.203,A -85,B 0,C 180,E1 29586.384,E2 29586.384} C_VEL
LIN {X 0,Y 678.323,Z 995.224,A -85,B 0,C 180,E1 29585.72,E2 29585.72} C_VEL
LIN {X 0,Y 678.802,Z 973.766,A -85,B 0,C 180,E1 29585.207,E2 29585.207} C_VEL
LIN {X 0,Y 679.173,Z 951.384,A -85,B 0,C 180,E1 29584.834,E2 29584.834} C_VEL
LIN {X 0,Y 681.38,Z 696.643,A -85,B 0,C 180,E1 29581.886,E2 29581.886} C_VEL
LIN {X 0,Y 681.432,Z 663.983,A -85,B 0,C 180,E1 29581.498,E2 29581.498} C_VEL
LIN {X 0,Y 678.81,Z 649.044,A -85,B 0,C 180,E1 29581.158,E2 29581.158} C_VEL
LIN {X 0,Y 680.167,Z 604.09,A -85,B 0,C 180,E1 29578.339,E2 29578.339} C_VEL
LIN {X 0,Y 681.798,Z 557.139,A -85,B 0,C 180,E1 29575.319,E2 29575.319} C_VEL
LIN {X 0,Y 683.256,Z 516.388,A -85,B 0,C 180,E1 29572.621,E2 29572.621} C_VEL
LIN {X 0,Y 674.909,Z 495.635,A -85,B 0,C 180,E1 29570.589,E2 29570.589} C_VEL
LIN {X 0,Y 672.616,Z 489.633,A -85,B 0,C 180,E1 29569.953,E2 29569.953} C_VEL
LIN {X 0,Y 672.552,Z 489.428,A -85,B 0,C 180,E1 29566.97,E2 29566.97} C_VEL
LIN {X 0,Y 672.581,Z 489.438,A -85,B 0,C 180,E1 29563.969,E2 29563.969} C_VEL
LIN {X 0,Y 672.547,Z 489.449,A -85,B 0,C 180,E1 29560.955,E2 29560.955} C_VEL
LIN {X 0,Y 672.578,Z 489.425,A -85,B 0,C 180,E1 29557.987,E2 29557.987} C_VEL
LIN {X 0,Y 672.55,Z 489.451,A -85,B 0,C 180,E1 29555,E2 29555} C_VEL
LIN {X 0,Y 672.583,Z 489.455,A -85,B 0,C 180,E1 29552.055,E2 29552.055} C_VEL
LIN {X 0,Y 672.558,Z 489.448,A -85,B 0,C 180,E1 29548.991,E2 29548.991} C_VEL
LIN {X 0,Y 672.577,Z 489.447,A -85,B 0,C 180,E1 29546.012,E2 29546.012} C_VEL
LIN {X 0,Y 672.556,Z 489.44,A -85,B 0,C 180,E1 29542.832,E2 29542.832} C_VEL
LIN {X 0,Y 672.569,Z 489.452,A -85,B 0,C 180,E1 29539.904,E2 29539.904} C_VEL
LIN {X 0,Y 672.566,Z 489.446,A -85,B 0,C 180,E1 29536.763,E2 29536.763} C_VEL
LIN {X 0,Y 672.564,Z 489.446,A -85,B 0,C 180,E1 29533.761,E2 29533.761} C_VEL
LIN {X 0,Y 672.558,Z 489.438,A -85,B 0,C 180,E1 29530.537,E2 29530.537} C_VEL
LIN {X 0,Y 672.56,Z 489.455,A -85,B 0,C 180,E1 29527.603,E2 29527.603} C_VEL
LIN {X 0,Y 672.566,Z 489.445,A -85,B 0,C 180,E1 29524.434,E2 29524.434} C_VEL
LIN {X 0,Y 672.548,Z 489.451,A -85,B 0,C 180,E1 29521.533,E2 29521.533} C_VEL
LIN {X 0,Y 672.583,Z 489.445,A -85,B 0,C 180,E1 29518.467,E2 29518.467} C_VEL
LIN {X 0,Y 672.538,Z 489.445,A -85,B 0,C 180,E1 29515.566,E2 29515.566} C_VEL
LIN {X 0,Y 672.585,Z 489.439,A -85,B 0,C 180,E1 29512.569,E2 29512.569} C_VEL
LIN {X 0,Y 672.539,Z 489.45,A -85,B 0,C 180,E1 29509.636,E2 29509.636} C_VEL
LIN {X 0,Y 672.585,Z 489.446,A -85,B 0,C 180,E1 29506.678,E2 29506.678} C_VEL
LIN {X 0,Y 672.547,Z 489.443,A -85,B 0,C 180,E1 29503.681,E2 29503.681} C_VEL
LIN {X 0,Y 672.554,Z 489.454,A -85,B 0,C 180,E1 29500.818,E2 29500.818} C_VEL
LIN {X 0,Y 672.556,Z 489.448,A -85,B 0,C 180,E1 29497.623,E2 29497.623} C_VEL
LIN {X 0,Y 672.537,Z 489.446,A -85,B 0,C 180,E1 29494.836,E2 29494.836} C_VEL
LIN {X 0,Y 672.589,Z 489.442,A -85,B 0,C 180,E1 29491.787,E2 29491.787} C_VEL
LIN {X 0,Y 672.531,Z 489.451,A -85,B 0,C 180,E1 29488.908,E2 29488.908} C_VEL
LIN {X 0,Y 672.583,Z 489.426,A -85,B 0,C 180,E1 29486.015,E2 29486.015} C_VEL
LIN {X 0,Y 672.535,Z 489.451,A -85,B 0,C 180,E1 29482.973,E2 29482.973} C_VEL
LIN {X 0,Y 672.551,Z 489.43,A -85,B 0,C 180,E1 29480.15,E2 29480.15} C_VEL
LIN {X 0,Y 672.545,Z 489.437,A -85,B 0,C 180,E1 29476.968,E2 29476.968} C_VEL
LIN {X 0,Y 672.535,Z 489.457,A -85,B 0,C 180,E1 29474.208,E2 29474.208} C_VEL
LIN {X 0,Y 672.579,Z 489.435,A -85,B 0,C 180,E1 29471.085,E2 29471.085} C_VEL
LIN {X 0,Y 672.559,Z 489.685,A -85,B 0,C 180,E1 29470.362,E2 29470.362} C_VEL
LIN {X 0,Y 674.665,Z 495.042,A -85,B 0,C 180,E1 29469.809,E2 29469.809} C_VEL
LIN {X 0,Y 683.824,Z 517.054,A -85,B 0,C 180,E1 29467.728,E2 29467.728} C_VEL
LIN {X 0,Y 683.401,Z 529.61,A -85,B 0,C 180,E1 29466.947,E2 29466.947} C_VEL
LIN {X 0,Y 686.842,Z 546.824,A -85,B 0,C 180,E1 29466.535,E2 29466.535} C_VEL
LIN {X 0,Y 685.325,Z 744.898,A -85,B 0,C 180,E1 29464.199,E2 29464.199} C_VEL
LIN {X 0,Y 683.705,Z 919.19,A -85,B 0,C 180,E1 29462.121,E2 29462.121} C_VEL
LIN {X 0,Y 683.104,Z 944.677,A -85,B 0,C 180,E1 29461.669,E2 29461.669} C_VEL
LIN {X 0,Y 682.426,Z 966.159,A -85,B 0,C 180,E1 29461.151,E2 29461.151} C_VEL
LIN {X 0,Y 681.657,Z 989.297,A -85,B 0,C 180,E1 29460.45,E2 29460.45} C_VEL
LIN {X 0,Y 680.783,Z 1010.242,A -85,B 0,C 180,E1 29459.666,E2 29459.666} C_VEL
LIN {X 0,Y 679.886,Z 1030.282,A -85,B 0,C 180,E1 29458.793,E2 29458.793} C_VEL
LIN {X 0,Y 678.73,Z 1053.523,A -85,B 0,C 180,E1 29457.6,E2 29457.6} C_VEL
LIN {X 0,Y 677.78,Z 1072.747,A -85,B 0,C 180,E1 29456.456,E2 29456.456} C_VEL
LIN {X 0,Y 676.661,Z 1094.021,A -85,B 0,C 180,E1 29454.999,E2 29454.999} C_VEL
LIN {X 0,Y 675.801,Z 1111.41,A -85,B 0,C 180,E1 29453.637,E2 29453.637} C_VEL
LIN {X 0,Y 674.847,Z 1130.614,A -85,B 0,C 180,E1 29451.923,E2 29451.923} C_VEL
LIN {X 0,Y 674.159,Z 1145.748,A -85,B 0,C 180,E1 29450.386,E2 29450.386} C_VEL
LIN {X 0,Y 673.468,Z 1161.822,A -85,B 0,C 180,E1 29448.525,E2 29448.525} C_VEL
LIN {X 0,Y 673,Z 1174.53,A -85,B 0,C 180,E1 29446.84,E2 29446.84} C_VEL
LIN {X 0,Y 672.581,Z 1187.767,A -85,B 0,C 180,E1 29444.815,E2 29444.815} C_VEL
LIN {X 0,Y 672.315,Z 1197.606,A -85,B 0,C 180,E1 29443.058,E2 29443.058} C_VEL
LIN {X 0,Y 672.101,Z 1207.478,A -85,B 0,C 180,E1 29440.977,E2 29440.977} C_VEL
LIN {X 0,Y 672.008,Z 1214.515,A -85,B 0,C 180,E1 29439.161,E2 29439.161} C_VEL
LIN {X 0,Y 671.934,Z 1220.508,A -85,B 0,C 180,E1 29437.266,E2 29437.266} C_VEL
LIN {X 0,Y 671.893,Z 1225.337,A -85,B 0,C 180,E1 29435.208,E2 29435.208} C_VEL
LIN {X 0,Y 671.908,Z 1228.237,A -85,B 0,C 180,E1 29433.412,E2 29433.412} C_VEL
LIN {X 0,Y 671.907,Z 1230.17,A -85,B 0,C 180,E1 29431.279,E2 29431.279} C_VEL
LIN {X 0,Y 671.882,Z 1230.351,A -85,B 0,C 180,E1 29429.403,E2 29429.403} C_VEL
LIN {X 0,Y 671.907,Z 1229.363,A -85,B 0,C 180,E1 29427.612,E2 29427.612} C_VEL
LIN {X 0,Y 671.918,Z 1226.45,A -85,B 0,C 180,E1 29425.391,E2 29425.391} C_VEL
LIN {X 0,Y 671.934,Z 1222.69,A -85,B 0,C 180,E1 29423.592,E2 29423.592} C_VEL
LIN {X 0,Y 671.993,Z 1217.202,A -85,B 0,C 180,E1 29421.616,E2 29421.616} C_VEL
LIN {X 0,Y 672.083,Z 1209.606,A -85,B 0,C 180,E1 29419.543,E2 29419.543} C_VEL
LIN {X 0,Y 672.225,Z 1201.528,A -85,B 0,C 180,E1 29417.72,E2 29417.72} C_VEL
LIN {X 0,Y 672.5,Z 1190.357,A -85,B 0,C 180,E1 29415.624,E2 29415.624} C_VEL
LIN {X 0,Y 672.839,Z 1179.392,A -85,B 0,C 180,E1 29413.866,E2 29413.866} C_VEL
LIN {X 0,Y 673.363,Z 1164.942,A -85,B 0,C 180,E1 29411.87,E2 29411.87} C_VEL
LIN {X 0,Y 673.944,Z 1150.698,A -85,B 0,C 180,E1 29410.158,E2 29410.158} C_VEL
LIN {X 0,Y 674.675,Z 1134.319,A -85,B 0,C 180,E1 29408.437,E2 29408.437} C_VEL
LIN {X 0,Y 675.453,Z 1118.136,A -85,B 0,C 180,E1 29406.935,E2 29406.935} C_VEL
LIN {X 0,Y 676.435,Z 1098.881,A -85,B 0,C 180,E1 29405.365,E2 29405.365} C_VEL
LIN {X 0,Y 677.325,Z 1081.086,A -85,B 0,C 180,E1 29404.091,E2 29404.091} C_VEL
LIN {X 0,Y 678.49,Z 1058.876,A -85,B 0,C 180,E1 29402.704,E2 29402.704} C_VEL
LIN {X 0,Y 679.434,Z 1039.328,A -85,B 0,C 180,E1 29401.649,E2 29401.649} C_VEL
LIN {X 0,Y 680.536,Z 1015.892,A -85,B 0,C 180,E1 29400.564,E2 29400.564} C_VEL
LIN {X 0,Y 681.38,Z 995.719,A -85,B 0,C 180,E1 29399.78,E2 29399.78} C_VEL
LIN {X 0,Y 682.246,Z 973.189,A -85,B 0,C 180,E1 29399.042,E2 29399.042} C_VEL
LIN {X 0,Y 682.938,Z 949.168,A -85,B 0,C 180,E1 29398.429,E2 29398.429} C_VEL
LIN {X 0,Y 683.572,Z 926.459,A -85,B 0,C 180,E1 29397.989,E2 29397.989} C_VEL
LIN {X 0,Y 684.017,Z 893.006,A -85,B 0,C 180,E1 29397.55,E2 29397.55} C_VEL
LIN {X 0,Y 686.089,Z 652.856,A -85,B 0,C 180,E1 29394.704,E2 29394.704} C_VEL
LIN {X 0,Y 686.671,Z 544.975,A -85,B 0,C 180,E1 29393.433,E2 29393.433} C_VEL
LIN {X 0,Y 683.39,Z 529.263,A -85,B 0,C 180,E1 29393.035,E2 29393.035} C_VEL
LIN {X 0,Y 683.672,Z 516.585,A -85,B 0,C 180,E1 29392.232,E2 29392.232} C_VEL
LIN {X 0,Y 673.759,Z 492.82,A -85,B 0,C 180,E1 29389.976,E2 29389.976} C_VEL
LIN {X 0,Y 672.553,Z 489.653,A -85,B 0,C 180,E1 29389.623,E2 29389.623} C_VEL
LIN {X 0,Y 672.563,Z 489.436,A -85,B 0,C 180,E1 29386.971,E2 29386.971} C_VEL
LIN {X 0,Y 672.541,Z 489.431,A -85,B 0,C 180,E1 29383.854,E2 29383.854} C_VEL
LIN {X 0,Y 672.539,Z 489.453,A -85,B 0,C 180,E1 29381.082,E2 29381.082} C_VEL
LIN {X 0,Y 672.577,Z 489.433,A -85,B 0,C 180,E1 29377.987,E2 29377.987} C_VEL
LIN {X 0,Y 672.531,Z 489.447,A -85,B 0,C 180,E1 29375.126,E2 29375.126} C_VEL
LIN {X 0,Y 672.585,Z 489.429,A -85,B 0,C 180,E1 29372.156,E2 29372.156} C_VEL
LIN {X 0,Y 672.535,Z 489.448,A -85,B 0,C 180,E1 29369.187,E2 29369.187} C_VEL
LIN {X 0,Y 672.577,Z 489.448,A -85,B 0,C 180,E1 29366.297,E2 29366.297} C_VEL
LIN {X 0,Y 672.546,Z 489.454,A -85,B 0,C 180,E1 29363.203,E2 29363.203} C_VEL
LIN {X 0,Y 672.553,Z 489.443,A -85,B 0,C 180,E1 29360.358,E2 29360.358} C_VEL
LIN {X 0,Y 672.566,Z 489.446,A -85,B 0,C 180,E1 29357.209,E2 29357.209} C_VEL
LIN {X 0,Y 672.547,Z 489.448,A -85,B 0,C 180,E1 29354.288,E2 29354.288} C_VEL
LIN {X 0,Y 672.578,Z 489.452,A -85,B 0,C 180,E1 29351.14,E2 29351.14} C_VEL
LIN {X 0,Y 672.543,Z 489.438,A -85,B 0,C 180,E1 29348.206,E2 29348.206} C_VEL
LIN {X 0,Y 672.584,Z 489.452,A -85,B 0,C 180,E1 29345.203,E2 29345.203} C_VEL
LIN {X 0,Y 672.541,Z 489.449,A -85,B 0,C 180,E1 29342.215,E2 29342.215} C_VEL
LIN {X 0,Y 672.584,Z 489.443,A -85,B 0,C 180,E1 29339.319,E2 29339.319} C_VEL
LIN {X 0,Y 672.547,Z 489.451,A -85,B 0,C 180,E1 29336.249,E2 29336.249} C_VEL
LIN {X 0,Y 672.586,Z 489.439,A -85,B 0,C 180,E1 29333.255,E2 29333.255} C_VEL
LIN {X 0,Y 672.553,Z 489.443,A -85,B 0,C 180,E1 29330.156,E2 29330.156} C_VEL
LIN {X 0,Y 672.579,Z 489.446,A -85,B 0,C 180,E1 29327.202,E2 29327.202} C_VEL
LIN {X 0,Y 672.56,Z 489.454,A -85,B 0,C 180,E1 29324.036,E2 29324.036} C_VEL
LIN {X 0,Y 672.581,Z 489.438,A -85,B 0,C 180,E1 29320.999,E2 29320.999} C_VEL
LIN {X 0,Y 672.562,Z 489.446,A -85,B 0,C 180,E1 29317.846,E2 29317.846} C_VEL
LIN {X 0,Y 672.581,Z 489.446,A -85,B 0,C 180,E1 29314.838,E2 29314.838} C_VEL
LIN {X 0,Y 672.566,Z 489.454,A -85,B 0,C 180,E1 29311.689,E2 29311.689} C_VEL
LIN {X 0,Y 672.586,Z 489.444,A -85,B 0,C 180,E1 29308.646,E2 29308.646} C_VEL
LIN {X 0,Y 672.583,Z 489.442,A -85,B 0,C 180,E1 29306.468,E2 29306.468} C_VEL
LIN {X 0,Y 671.6,Z 489.572,A -85,B 0,C 180,E1 29305.812,E2 29305.812} C_VEL
LIN {X 0,Y 665.184,Z 490.369,A -85,B 0,C 180,E1 29303.973,E2 29303.973} C_VEL
LIN {X 0,Y 664.63,Z 490.425,A -85,B 0,C 180,E1 29303.495,E2 29303.495} C_VEL
LIN {X 0,Y 664.648,Z 490.431,A -85,B 0,C 180,E1 29300.367,E2 29300.367} C_VEL
LIN {X 0,Y 664.625,Z 490.415,A -85,B 0,C 180,E1 29297.235,E2 29297.235} C_VEL
LIN {X 0,Y 664.645,Z 490.433,A -85,B 0,C 180,E1 29294.143,E2 29294.143} C_VEL
LIN {X 0,Y 664.629,Z 490.445,A -85,B 0,C 180,E1 29290.989,E2 29290.989} C_VEL
LIN {X 0,Y 664.676,Z 490.784,A -85,B 0,C 180,E1 29290.426,E2 29290.426} C_VEL
LIN {X 0,Y 674.461,Z 514.92,A -85,B 0,C 180,E1 29287.968,E2 29287.968} C_VEL
LIN {X 0,Y 676.364,Z 520.445,A -85,B 0,C 180,E1 29287.451,E2 29287.451} C_VEL
LIN {X 0,Y 674.506,Z 565.71,A -85,B 0,C 180,E1 29284.438,E2 29284.438} C_VEL
LIN {X 0,Y 672.813,Z 611.278,A -85,B 0,C 180,E1 29281.486,E2 29281.486} C_VEL
LIN {X 0,Y 671.657,Z 649.071,A -85,B 0,C 180,E1 29279.114,E2 29279.114} C_VEL
LIN {X 0,Y 674.83,Z 667.627,A -85,B 0,C 180,E1 29278.72,E2 29278.72} C_VEL
LIN {X 0,Y 672.654,Z 915.439,A -85,B 0,C 180,E1 29275.85,E2 29275.85} C_VEL
LIN {X 0,Y 672.144,Z 958.296,A -85,B 0,C 180,E1 29275.32,E2 29275.32} C_VEL
LIN {X 0,Y 671.571,Z 979.681,A -85,B 0,C 180,E1 29274.899,E2 29274.899} C_VEL
LIN {X 0,Y 670.89,Z 1001.203,A -85,B 0,C 180,E1 29274.312,E2 29274.312} C_VEL
LIN {X 0,Y 670.096,Z 1022.543,A -85,B 0,C 180,E1 29273.571,E2 29273.571} C_VEL
LIN {X 0,Y 669.373,Z 1041.779,A -85,B 0,C 180,E1 29272.76,E2 29272.76} C_VEL
LIN {X 0,Y 668.543,Z 1061.651,A -85,B 0,C 180,E1 29271.753,E2 29271.753} C_VEL
LIN {X 0,Y 667.743,Z 1080.406,A -85,B 0,C 180,E1 29270.627,E2 29270.627} C_VEL
LIN {X 0,Y 666.979,Z 1097.922,A -85,B 0,C 180,E1 29269.393,E2 29269.393} C_VEL
LIN {X 0,Y 666.256,Z 1114.177,A -85,B 0,C 180,E1 29268.053,E2 29268.053} C_VEL
LIN {X 0,Y 665.627,Z 1129.597,A -85,B 0,C 180,E1 29266.583,E2 29266.583} C_VEL
LIN {X 0,Y 665.1,Z 1143.99,A -85,B 0,C 180,E1 29264.985,E2 29264.985} C_VEL
LIN {X 0,Y 664.67,Z 1156.764,A -85,B 0,C 180,E1 29263.306,E2 29263.306} C_VEL
LIN {X 0,Y 664.35,Z 1168.063,A -85,B 0,C 180,E1 29261.547,E2 29261.547} C_VEL
LIN {X 0,Y 664.146,Z 1177.457,A -85,B 0,C 180,E1 29259.795,E2 29259.795} C_VEL
LIN {X 0,Y 664.026,Z 1185.049,A -85,B 0,C 180,E1 29258.05,E2 29258.05} C_VEL
LIN {X 0,Y 663.95,Z 1191.271,A -85,B 0,C 180,E1 29256.225,E2 29256.225} C_VEL
LIN {X 0,Y 663.926,Z 1195.899,A -85,B 0,C 180,E1 29254.405,E2 29254.405} C_VEL
LIN {X 0,Y 663.914,Z 1198.842,A -85,B 0,C 180,E1 29252.59,E2 29252.59} C_VEL
LIN {X 0,Y 663.905,Z 1200.335,A -85,B 0,C 180,E1 29250.604,E2 29250.604} C_VEL
LIN {X 0,Y 663.904,Z 1200.184,A -85,B 0,C 180,E1 29248.792,E2 29248.792} C_VEL
LIN {X 0,Y 663.911,Z 1198.394,A -85,B 0,C 180,E1 29246.979,E2 29246.979} C_VEL
LIN {X 0,Y 663.918,Z 1194.921,A -85,B 0,C 180,E1 29245.076,E2 29245.076} C_VEL
LIN {X 0,Y 663.951,Z 1190.008,A -85,B 0,C 180,E1 29243.254,E2 29243.254} C_VEL
LIN {X 0,Y 664.048,Z 1183.294,A -85,B 0,C 180,E1 29241.427,E2 29241.427} C_VEL
LIN {X 0,Y 664.208,Z 1174.372,A -85,B 0,C 180,E1 29239.505,E2 29239.505} C_VEL
LIN {X 0,Y 664.445,Z 1164.404,A -85,B 0,C 180,E1 29237.75,E2 29237.75} C_VEL
LIN {X 0,Y 664.782,Z 1152.962,A -85,B 0,C 180,E1 29236.075,E2 29236.075} C_VEL
LIN {X 0,Y 665.231,Z 1140.033,A -85,B 0,C 180,E1 29234.467,E2 29234.467} C_VEL
LIN {X 0,Y 665.779,Z 1126.116,A -85,B 0,C 180,E1 29232.971,E2 29232.971} C_VEL
LIN {X 0,Y 666.425,Z 1110.62,A -85,B 0,C 180,E1 29231.544,E2 29231.544} C_VEL
LIN {X 0,Y 667.143,Z 1093.651,A -85,B 0,C 180,E1 29230.202,E2 29230.202} C_VEL
LIN {X 0,Y 667.971,Z 1075.112,A -85,B 0,C 180,E1 29228.946,E2 29228.946} C_VEL
LIN {X 0,Y 668.793,Z 1056.413,A -85,B 0,C 180,E1 29227.868,E2 29227.868} C_VEL
LIN {X 0,Y 669.526,Z 1037.698,A -85,B 0,C 180,E1 29226.967,E2 29226.967} C_VEL
LIN {X 0,Y 670.33,Z 1015.86,A -85,B 0,C 180,E1 29226.094,E2 29226.094} C_VEL
LIN {X 0,Y 671.093,Z 996.079,A -85,B 0,C 180,E1 29225.438,E2 29225.438} C_VEL
LIN {X 0,Y 671.718,Z 974.866,A -85,B 0,C 180,E1 29224.904,E2 29224.904} C_VEL
LIN {X 0,Y 672.233,Z 952.396,A -85,B 0,C 180,E1 29224.505,E2 29224.505} C_VEL
LIN {X 0,Y 674.067,Z 756.504,A -85,B 0,C 180,E1 29222.213,E2 29222.213} C_VEL
LIN {X 0,Y 674.65,Z 665.387,A -85,B 0,C 180,E1 29221.154,E2 29221.154} C_VEL
LIN {X 0,Y 671.587,Z 648.337,A -85,B 0,C 180,E1 29220.769,E2 29220.769} C_VEL
LIN {X 0,Y 673.138,Z 602.375,A -85,B 0,C 180,E1 29217.854,E2 29217.854} C_VEL
LIN {X 0,Y 674.858,Z 557.175,A -85,B 0,C 180,E1 29214.911,E2 29214.911} C_VEL
LIN {X 0,Y 676.335,Z 519.833,A -85,B 0,C 180,E1 29212.413,E2 29212.413} C_VEL
LIN {X 0,Y 667.527,Z 497.655,A -85,B 0,C 180,E1 29210.213,E2 29210.213} C_VEL
LIN {X 0,Y 664.65,Z 490.671,A -85,B 0,C 180,E1 29209.454,E2 29209.454} C_VEL
LIN {X 0,Y 664.64,Z 490.414,A -85,B 0,C 180,E1 29206.568,E2 29206.568} C_VEL
LIN {X 0,Y 664.622,Z 490.419,A -85,B 0,C 180,E1 29203.435,E2 29203.435} C_VEL
LIN {X 0,Y 664.643,Z 490.444,A -85,B 0,C 180,E1 29200.421,E2 29200.421} C_VEL
LIN {X 0,Y 664.621,Z 490.417,A -85,B 0,C 180,E1 29197.267,E2 29197.267} C_VEL
LIN {X 0,Y 664.64,Z 490.44,A -85,B 0,C 180,E1 29194.239,E2 29194.239} C_VEL
LIN {X 0,Y 664.62,Z 490.436,A -85,B 0,C 180,E1 29191.066,E2 29191.066} C_VEL
LIN {X 0,Y 664.636,Z 490.445,A -85,B 0,C 180,E1 29188.092,E2 29188.092} C_VEL
LIN {X 0,Y 664.62,Z 490.437,A -85,B 0,C 180,E1 29184.914,E2 29184.914} C_VEL
LIN {X 0,Y 664.636,Z 490.436,A -85,B 0,C 180,E1 29181.907,E2 29181.907} C_VEL
LIN {X 0,Y 664.623,Z 490.428,A -85,B 0,C 180,E1 29178.781,E2 29178.781} C_VEL
LIN {X 0,Y 664.627,Z 490.442,A -85,B 0,C 180,E1 29175.801,E2 29175.801} C_VEL
LIN {X 0,Y 664.622,Z 490.436,A -85,B 0,C 180,E1 29172.6,E2 29172.6} C_VEL
LIN {X 0,Y 664.625,Z 490.433,A -85,B 0,C 180,E1 29169.613,E2 29169.613} C_VEL
LIN {X 0,Y 664.625,Z 490.429,A -85,B 0,C 180,E1 29166.479,E2 29166.479} C_VEL
LIN {X 0,Y 664.616,Z 490.442,A -85,B 0,C 180,E1 29163.536,E2 29163.536} C_VEL
LIN {X 0,Y 664.629,Z 490.432,A -85,B 0,C 180,E1 29160.345,E2 29160.345} C_VEL
LIN {X 0,Y 664.609,Z 490.442,A -85,B 0,C 180,E1 29157.413,E2 29157.413} C_VEL
LIN {X 0,Y 664.641,Z 490.435,A -85,B 0,C 180,E1 29154.302,E2 29154.302} C_VEL
LIN {X 0,Y 664.602,Z 490.431,A -85,B 0,C 180,E1 29151.347,E2 29151.347} C_VEL
LIN {X 0,Y 664.646,Z 490.429,A -85,B 0,C 180,E1 29148.282,E2 29148.282} C_VEL
LIN {X 0,Y 664.595,Z 490.441,A -85,B 0,C 180,E1 29145.322,E2 29145.322} C_VEL
LIN {X 0,Y 664.648,Z 490.436,A -85,B 0,C 180,E1 29142.399,E2 29142.399} C_VEL
LIN {X 0,Y 664.597,Z 490.433,A -85,B 0,C 180,E1 29139.353,E2 29139.353} C_VEL
LIN {X 0,Y 664.636,Z 490.443,A -85,B 0,C 180,E1 29136.505,E2 29136.505} C_VEL
LIN {X 0,Y 664.604,Z 490.439,A -85,B 0,C 180,E1 29133.334,E2 29133.334} C_VEL
LIN {X 0,Y 664.611,Z 490.439,A -85,B 0,C 180,E1 29130.53,E2 29130.53} C_VEL
LIN {X 0,Y 664.613,Z 490.414,A -85,B 0,C 180,E1 29127.309,E2 29127.309} C_VEL
LIN {X 0,Y 664.6,Z 490.439,A -85,B 0,C 180,E1 29124.479,E2 29124.479} C_VEL
LIN {X 0,Y 664.633,Z 490.408,A -85,B 0,C 180,E1 29121.331,E2 29121.331} C_VEL
LIN {X 0,Y 664.593,Z 490.445,A -85,B 0,C 180,E1 29118.433,E2 29118.433} C_VEL
LIN {X 0,Y 664.645,Z 490.419,A -85,B 0,C 180,E1 29115.362,E2 29115.362} C_VEL
LIN {X 0,Y 664.586,Z 490.418,A -85,B 0,C 180,E1 29112.494,E2 29112.494} C_VEL
LIN {X 0,Y 664.649,Z 490.688,A -85,B 0,C 180,E1 29110.863,E2 29110.863} C_VEL
LIN {X 0,Y 667.341,Z 497.349,A -85,B 0,C 180,E1 29110.169,E2 29110.169} C_VEL
LIN {X 0,Y 676.938,Z 520.404,A -85,B 0,C 180,E1 29107.952,E2 29107.952} C_VEL
LIN {X 0,Y 676.667,Z 531.115,A -85,B 0,C 180,E1 29107.3,E2 29107.3} C_VEL
LIN {X 0,Y 680.119,Z 548.348,A -85,B 0,C 180,E1 29106.885,E2 29106.885} C_VEL
LIN {X 0,Y 678.108,Z 803.002,A -85,B 0,C 180,E1 29103.886,E2 29103.886} C_VEL
LIN {X 0,Y 676.918,Z 919.595,A -85,B 0,C 180,E1 29102.477,E2 29102.477} C_VEL
LIN {X 0,Y 676.258,Z 945.066,A -85,B 0,C 180,E1 29102.018,E2 29102.018} C_VEL
LIN {X 0,Y 675.533,Z 966.276,A -85,B 0,C 180,E1 29101.501,E2 29101.501} C_VEL
LIN {X 0,Y 674.677,Z 989.293,A -85,B 0,C 180,E1 29100.799,E2 29100.799} C_VEL
LIN {X 0,Y 673.724,Z 1010.238,A -85,B 0,C 180,E1 29100.009,E2 29100.009} C_VEL
LIN {X 0,Y 672.745,Z 1030.297,A -85,B 0,C 180,E1 29099.127,E2 29099.127} C_VEL
LIN {X 0,Y 671.474,Z 1053.52,A -85,B 0,C 180,E1 29097.924,E2 29097.924} C_VEL
LIN {X 0,Y 670.428,Z 1072.747,A -85,B 0,C 180,E1 29096.769,E2 29096.769} C_VEL
LIN {X 0,Y 669.207,Z 1094.018,A -85,B 0,C 180,E1 29095.297,E2 29095.297} C_VEL
LIN {X 0,Y 668.24,Z 1111.411,A -85,B 0,C 180,E1 29093.921,E2 29093.921} C_VEL
LIN {X 0,Y 667.193,Z 1130.614,A -85,B 0,C 180,E1 29092.188,E2 29092.188} C_VEL
LIN {X 0,Y 666.423,Z 1145.64,A -85,B 0,C 180,E1 29090.645,E2 29090.645} C_VEL
LIN {X 0,Y 665.653,Z 1161.823,A -85,B 0,C 180,E1 29088.75,E2 29088.75} C_VEL
LIN {X 0,Y 665.138,Z 1174.556,A -85,B 0,C 180,E1 29087.041,E2 29087.041} C_VEL
LIN {X 0,Y 664.665,Z 1187.768,A -85,B 0,C 180,E1 29084.995,E2 29084.995} C_VEL
LIN {X 0,Y 664.356,Z 1197.945,A -85,B 0,C 180,E1 29083.151,E2 29083.151} C_VEL
LIN {X 0,Y 664.117,Z 1207.957,A -85,B 0,C 180,E1 29080.992,E2 29080.992} C_VEL
LIN {X 0,Y 664.018,Z 1214.818,A -85,B 0,C 180,E1 29079.184,E2 29079.184} C_VEL
LIN {X 0,Y 663.943,Z 1221.016,A -85,B 0,C 180,E1 29077.18,E2 29077.18} C_VEL
LIN {X 0,Y 663.894,Z 1225.497,A -85,B 0,C 180,E1 29075.184,E2 29075.184} C_VEL
LIN {X 0,Y 663.905,Z 1228.35,A -85,B 0,C 180,E1 29073.367,E2 29073.367} C_VEL
LIN {X 0,Y 663.91,Z 1230.193,A -85,B 0,C 180,E1 29071.208,E2 29071.208} C_VEL
LIN {X 0,Y 663.884,Z 1230.328,A -85,B 0,C 180,E1 29069.31,E2 29069.31} C_VEL
LIN {X 0,Y 663.891,Z 1229.226,A -85,B 0,C 180,E1 29067.41,E2 29067.41} C_VEL
LIN {X 0,Y 663.911,Z 1226.291,A -85,B 0,C 180,E1 29065.249,E2 29065.249} C_VEL
LIN {X 0,Y 663.937,Z 1222.484,A -85,B 0,C 180,E1 29063.428,E2 29063.428} C_VEL
LIN {X 0,Y 663.99,Z 1216.636,A -85,B 0,C 180,E1 29061.339,E2 29061.339} C_VEL
LIN {X 0,Y 664.109,Z 1209.253,A -85,B 0,C 180,E1 29059.328,E2 29059.328} C_VEL
LIN {X 0,Y 664.313,Z 1200.305,A -85,B 0,C 180,E1 29057.306,E2 29057.306} C_VEL
LIN {X 0,Y 664.596,Z 1189.673,A -85,B 0,C 180,E1 29055.331,E2 29055.331} C_VEL
LIN {X 0,Y 664.993,Z 1178.235,A -85,B 0,C 180,E1 29053.491,E2 29053.491} C_VEL
LIN {X 0,Y 665.546,Z 1164.632,A -85,B 0,C 180,E1 29051.61,E2 29051.61} C_VEL
LIN {X 0,Y 666.197,Z 1150.534,A -85,B 0,C 180,E1 29049.898,E2 29049.898} C_VEL
LIN {X 0,Y 667.03,Z 1133.642,A -85,B 0,C 180,E1 29048.109,E2 29048.109} C_VEL
LIN {X 0,Y 667.911,Z 1117.395,A -85,B 0,C 180,E1 29046.591,E2 29046.591} C_VEL
LIN {X 0,Y 668.993,Z 1097.665,A -85,B 0,C 180,E1 29044.978,E2 29044.978} C_VEL
LIN {X 0,Y 670.116,Z 1078.411,A -85,B 0,C 180,E1 29043.6,E2 29043.6} C_VEL
LIN {X 0,Y 671.264,Z 1057.571,A -85,B 0,C 180,E1 29042.307,E2 29042.307} C_VEL
LIN {X 0,Y 672.321,Z 1037.873,A -85,B 0,C 180,E1 29041.243,E2 29041.243} C_VEL
LIN {X 0,Y 673.517,Z 1014.763,A -85,B 0,C 180,E1 29040.177,E2 29040.177} C_VEL
LIN {X 0,Y 674.442,Z 994.43,A -85,B 0,C 180,E1 29039.387,E2 29039.387} C_VEL
LIN {X 0,Y 675.39,Z 970.716,A -85,B 0,C 180,E1 29038.618,E2 29038.618} C_VEL
LIN {X 0,Y 676.147,Z 947.937,A -85,B 0,C 180,E1 29038.045,E2 29038.045} C_VEL
LIN {X 0,Y 676.869,Z 923.825,A -85,B 0,C 180,E1 29037.583,E2 29037.583} C_VEL
LIN {X 0,Y 677.397,Z 878.571,A -85,B 0,C 180,E1 29037.015,E2 29037.015} C_VEL
LIN {X 0,Y 678.846,Z 707.624,A -85,B 0,C 180,E1 29035.002,E2 29035.002} C_VEL
LIN {X 0,Y 679.992,Z 546.742,A -85,B 0,C 180,E1 29033.088,E2 29033.088} C_VEL
LIN {X 0,Y 676.562,Z 530.213,A -85,B 0,C 180,E1 29032.666,E2 29032.666} C_VEL
LIN {X 0,Y 676.798,Z 520.06,A -85,B 0,C 180,E1 29032.016,E2 29032.016} C_VEL
LIN {X 0,Y 667.341,Z 497.349,A -85,B 0,C 180,E1 29029.831,E2 29029.831} C_VEL
LIN {X 0,Y 664.65,Z 490.698,A -85,B 0,C 180,E1 29029.139,E2 29029.139} C_VEL
LIN {X 0,Y 664.616,Z 490.422,A -85,B 0,C 180,E1 29027.039,E2 29027.039} C_VEL
LIN {X 0,Y 664.606,Z 490.417,A -85,B 0,C 180,E1 29023.894,E2 29023.894} C_VEL
LIN {X 0,Y 664.6,Z 490.442,A -85,B 0,C 180,E1 29021.086,E2 29021.086} C_VEL
LIN {X 0,Y 664.637,Z 490.42,A -85,B 0,C 180,E1 29017.974,E2 29017.974} C_VEL
LIN {X 0,Y 664.594,Z 490.435,A -85,B 0,C 180,E1 29015.072,E2 29015.072} C_VEL
LIN {X 0,Y 664.647,Z 490.417,A -85,B 0,C 180,E1 29012.077,E2 29012.077} C_VEL
LIN {X 0,Y 664.596,Z 490.437,A -85,B 0,C 180,E1 29009.174,E2 29009.174} C_VEL
LIN {X 0,Y 664.642,Z 490.437,A -85,B 0,C 180,E1 29006.251,E2 29006.251} C_VEL
LIN {X 0,Y 664.603,Z 490.443,A -85,B 0,C 180,E1 29003.121,E2 29003.121} C_VEL
LIN {X 0,Y 664.625,Z 490.431,A -85,B 0,C 180,E1 29000.244,E2 29000.244} C_VEL
LIN {X 0,Y 664.614,Z 490.435,A -85,B 0,C 180,E1 28997.06,E2 28997.06} C_VEL
LIN {X 0,Y 664.615,Z 490.437,A -85,B 0,C 180,E1 28994.195,E2 28994.195} C_VEL
LIN {X 0,Y 664.63,Z 490.444,A -85,B 0,C 180,E1 28991.015,E2 28991.015} C_VEL
LIN {X 0,Y 664.614,Z 490.425,A -85,B 0,C 180,E1 28988.043,E2 28988.043} C_VEL
LIN {X 0,Y 664.63,Z 490.436,A -85,B 0,C 180,E1 28984.833,E2 28984.833} C_VEL
LIN {X 0,Y 664.62,Z 490.435,A -85,B 0,C 180,E1 28981.81,E2 28981.81} C_VEL
LIN {X 0,Y 664.629,Z 490.435,A -85,B 0,C 180,E1 28978.621,E2 28978.621} C_VEL
LIN {X 0,Y 664.625,Z 490.435,A -85,B 0,C 180,E1 28975.6,E2 28975.6} C_VEL
LIN {X 0,Y 664.628,Z 490.444,A -85,B 0,C 180,E1 28972.392,E2 28972.392} C_VEL
LIN {X 0,Y 664.633,Z 490.425,A -85,B 0,C 180,E1 28969.336,E2 28969.336} C_VEL
LIN {X 0,Y 664.625,Z 490.434,A -85,B 0,C 180,E1 28966.16,E2 28966.16} C_VEL
LIN {X 0,Y 664.641,Z 490.434,A -85,B 0,C 180,E1 28963.091,E2 28963.091} C_VEL
LIN {X 0,Y 664.625,Z 490.443,A -85,B 0,C 180,E1 28959.939,E2 28959.939} C_VEL
LIN {X 0,Y 664.644,Z 490.426,A -85,B 0,C 180,E1 28956.88,E2 28956.88} C_VEL
LIN {X 0,Y 664.624,Z 490.435,A -85,B 0,C 180,E1 28953.717,E2 28953.717} C_VEL
LIN {X 0,Y 664.65,Z 490.434,A -85,B 0,C 180,E1 28950.631,E2 28950.631} C_VEL
LIN {X 0,Y 664.624,Z 490.439,A -85,B 0,C 180,E1 28947.514,E2 28947.514} C_VEL
LIN {X 0,Y 664.646,Z 490.436,A -85,B 0,C 180,E1 28944.474,E2 28944.474} C_VEL
LIN {X 0,Y 664.63,Z 490.425,A -85,B 0,C 180,E1 28943.495,E2 28943.495} C_VEL
LIN {X 0,Y 663.608,Z 490.544,A -85,B 0,C 180,E1 28942.831,E2 28942.831} C_VEL
LIN {X 0,Y 657.2,Z 491.356,A -85,B 0,C 180,E1 28940.969,E2 28940.969} C_VEL
LIN {X 0,Y 656.703,Z 491.421,A -85,B 0,C 180,E1 28940.485,E2 28940.485} C_VEL
LIN {X 0,Y 656.695,Z 491.401,A -85,B 0,C 180,E1 28937.341,E2 28937.341} C_VEL
LIN {X 0,Y 656.706,Z 491.42,A -85,B 0,C 180,E1 28934.181,E2 28934.181} C_VEL
LIN {X 0,Y 656.701,Z 491.512,A -85,B 0,C 180,E1 28931.012,E2 28931.012} C_VEL
LIN {X 0,Y 657.696,Z 494.443,A -85,B 0,C 180,E1 28930.656,E2 28930.656} C_VEL
LIN {X 0,Y 665.608,Z 513.464,A -85,B 0,C 180,E1 28928.675,E2 28928.675} C_VEL
LIN {X 0,Y 669.45,Z 523.891,A -85,B 0,C 180,E1 28927.664,E2 28927.664} C_VEL
LIN {X 0,Y 667.371,Z 570.313,A -85,B 0,C 180,E1 28924.546,E2 28924.546} C_VEL
LIN {X 0,Y 665.557,Z 615.533,A -85,B 0,C 180,E1 28921.589,E2 28921.589} C_VEL
LIN {X 0,Y 664.465,Z 648.152,A -85,B 0,C 180,E1 28919.523,E2 28919.523} C_VEL
LIN {X 0,Y 668.059,Z 668.862,A -85,B 0,C 180,E1 28919.073,E2 28919.073} C_VEL
LIN {X 0,Y 665.907,Z 909.768,A -85,B 0,C 180,E1 28916.28,E2 28916.28} C_VEL
LIN {X 0,Y 665.338,Z 957.812,A -85,B 0,C 180,E1 28915.69,E2 28915.69} C_VEL
LIN {X 0,Y 664.707,Z 979.346,A -85,B 0,C 180,E1 28915.266,E2 28915.266} C_VEL
LIN {X 0,Y 663.962,Z 1000.899,A -85,B 0,C 180,E1 28914.677,E2 28914.677} C_VEL
LIN {X 0,Y 663.118,Z 1020.918,A -85,B 0,C 180,E1 28913.981,E2 28913.981} C_VEL
LIN {X 0,Y 662.132,Z 1040.761,A -85,B 0,C 180,E1 28913.117,E2 28913.117} C_VEL
LIN {X 0,Y 661.082,Z 1060.65,A -85,B 0,C 180,E1 28912.077,E2 28912.077} C_VEL
LIN {X 0,Y 660.11,Z 1080.985,A -85,B 0,C 180,E1 28910.837,E2 28910.837} C_VEL
LIN {X 0,Y 659.277,Z 1098.535,A -85,B 0,C 180,E1 28909.583,E2 28909.583} C_VEL
LIN {X 0,Y 658.463,Z 1115.195,A -85,B 0,C 180,E1 28908.183,E2 28908.183} C_VEL
LIN {X 0,Y 657.776,Z 1130.446,A -85,B 0,C 180,E1 28906.696,E2 28906.696} C_VEL
LIN {X 0,Y 657.232,Z 1143.995,A -85,B 0,C 180,E1 28905.169,E2 28905.169} C_VEL
LIN {X 0,Y 656.752,Z 1156.767,A -85,B 0,C 180,E1 28903.47,E2 28903.47} C_VEL
LIN {X 0,Y 656.401,Z 1168.066,A -85,B 0,C 180,E1 28901.688,E2 28901.688} C_VEL
LIN {X 0,Y 656.175,Z 1177.46,A -85,B 0,C 180,E1 28899.915,E2 28899.915} C_VEL
LIN {X 0,Y 656.041,Z 1185.051,A -85,B 0,C 180,E1 28898.148,E2 28898.148} C_VEL
LIN {X 0,Y 655.956,Z 1191.272,A -85,B 0,C 180,E1 28896.301,E2 28896.301} C_VEL
LIN {X 0,Y 655.925,Z 1195.9,A -85,B 0,C 180,E1 28894.459,E2 28894.459} C_VEL
LIN {X 0,Y 655.914,Z 1198.843,A -85,B 0,C 180,E1 28892.621,E2 28892.621} C_VEL
LIN {X 0,Y 655.906,Z 1200.335,A -85,B 0,C 180,E1 28890.611,E2 28890.611} C_VEL
LIN {X 0,Y 655.903,Z 1200.184,A -85,B 0,C 180,E1 28888.777,E2 28888.777} C_VEL
LIN {X 0,Y 655.912,Z 1198.296,A -85,B 0,C 180,E1 28886.867,E2 28886.867} C_VEL
LIN {X 0,Y 655.924,Z 1194.713,A -85,B 0,C 180,E1 28884.928,E2 28884.928} C_VEL
LIN {X 0,Y 655.962,Z 1189.735,A -85,B 0,C 180,E1 28883.084,E2 28883.084} C_VEL
LIN {X 0,Y 656.066,Z 1182.939,A -85,B 0,C 180,E1 28881.234,E2 28881.234} C_VEL
LIN {X 0,Y 656.249,Z 1174.203,A -85,B 0,C 180,E1 28879.345,E2 28879.345} C_VEL
LIN {X 0,Y 656.511,Z 1164.399,A -85,B 0,C 180,E1 28877.6,E2 28877.6} C_VEL
LIN {X 0,Y 656.886,Z 1152.958,A -85,B 0,C 180,E1 28875.905,E2 28875.905} C_VEL
LIN {X 0,Y 657.369,Z 1140.161,A -85,B 0,C 180,E1 28874.292,E2 28874.292} C_VEL
LIN {X 0,Y 657.979,Z 1126.109,A -85,B 0,C 180,E1 28872.763,E2 28872.763} C_VEL
LIN {X 0,Y 658.701,Z 1110.409,A -85,B 0,C 180,E1 28871.302,E2 28871.302} C_VEL
LIN {X 0,Y 659.487,Z 1093.641,A -85,B 0,C 180,E1 28869.962,E2 28869.962} C_VEL
LIN {X 0,Y 660.386,Z 1075.099,A -85,B 0,C 180,E1 28868.693,E2 28868.693} C_VEL
LIN {X 0,Y 661.492,Z 1053.253,A -85,B 0,C 180,E1 28867.423,E2 28867.423} C_VEL
LIN {X 0,Y 662.485,Z 1033.894,A -85,B 0,C 180,E1 28866.472,E2 28866.472} C_VEL
LIN {X 0,Y 663.375,Z 1014.775,A -85,B 0,C 180,E1 28865.703,E2 28865.703} C_VEL
LIN {X 0,Y 664.22,Z 994.108,A -85,B 0,C 180,E1 28865.026,E2 28865.026} C_VEL
LIN {X 0,Y 664.91,Z 973.383,A -85,B 0,C 180,E1 28864.512,E2 28864.512} C_VEL
LIN {X 0,Y 665.432,Z 951.255,A -85,B 0,C 180,E1 28864.127,E2 28864.127} C_VEL
LIN {X 0,Y 667.32,Z 757.426,A -85,B 0,C 180,E1 28861.853,E2 28861.853} C_VEL
LIN {X 0,Y 667.873,Z 666.676,A -85,B 0,C 180,E1 28860.8,E2 28860.8} C_VEL
LIN {X 0,Y 664.399,Z 647.417,A -85,B 0,C 180,E1 28860.36,E2 28860.36} C_VEL
LIN {X 0,Y 666.156,Z 600.662,A -85,B 0,C 180,E1 28857.358,E2 28857.358} C_VEL
LIN {X 0,Y 668.013,Z 555.352,A -85,B 0,C 180,E1 28854.368,E2 28854.368} C_VEL
LIN {X 0,Y 669.423,Z 523.277,A -85,B 0,C 180,E1 28852.2,E2 28852.2} C_VEL
LIN {X 0,Y 661.051,Z 502.12,A -85,B 0,C 180,E1 28850.075,E2 28850.075} C_VEL
LIN {X 0,Y 656.734,Z 491.785,A -85,B 0,C 180,E1 28848.955,E2 28848.955} C_VEL
LIN {X 0,Y 656.701,Z 491.409,A -85,B 0,C 180,E1 28848.121,E2 28848.121} C_VEL
LIN {X 0,Y 656.673,Z 491.433,A -85,B 0,C 180,E1 28845.076,E2 28845.076} C_VEL
LIN {X 0,Y 656.7,Z 491.407,A -85,B 0,C 180,E1 28842.063,E2 28842.063} C_VEL
LIN {X 0,Y 656.672,Z 491.419,A -85,B 0,C 180,E1 28839.056,E2 28839.056} C_VEL
LIN {X 0,Y 656.704,Z 491.421,A -85,B 0,C 180,E1 28836.054,E2 28836.054} C_VEL
LIN {X 0,Y 656.674,Z 491.422,A -85,B 0,C 180,E1 28832.97,E2 28832.97} C_VEL
LIN {X 0,Y 656.712,Z 491.423,A -85,B 0,C 180,E1 28829.961,E2 28829.961} C_VEL
LIN {X 0,Y 656.676,Z 491.42,A -85,B 0,C 180,E1 28826.843,E2 28826.843} C_VEL
LIN {X 0,Y 656.708,Z 491.423,A -85,B 0,C 180,E1 28823.796,E2 28823.796} C_VEL
LIN {X 0,Y 656.674,Z 491.427,A -85,B 0,C 180,E1 28820.687,E2 28820.687} C_VEL
LIN {X 0,Y 656.706,Z 491.428,A -85,B 0,C 180,E1 28817.638,E2 28817.638} C_VEL
LIN {X 0,Y 656.674,Z 491.416,A -85,B 0,C 180,E1 28814.551,E2 28814.551} C_VEL
LIN {X 0,Y 656.695,Z 491.429,A -85,B 0,C 180,E1 28811.595,E2 28811.595} C_VEL
LIN {X 0,Y 656.677,Z 491.426,A -85,B 0,C 180,E1 28808.405,E2 28808.405} C_VEL
LIN {X 0,Y 656.694,Z 491.421,A -85,B 0,C 180,E1 28805.417,E2 28805.417} C_VEL
LIN {X 0,Y 656.678,Z 491.422,A -85,B 0,C 180,E1 28802.269,E2 28802.269} C_VEL
LIN {X 0,Y 656.687,Z 491.429,A -85,B 0,C 180,E1 28799.302,E2 28799.302} C_VEL
LIN {X 0,Y 656.674,Z 491.418,A -85,B 0,C 180,E1 28796.071,E2 28796.071} C_VEL
LIN {X 0,Y 656.687,Z 491.43,A -85,B 0,C 180,E1 28793.091,E2 28793.091} C_VEL
LIN {X 0,Y 656.676,Z 491.427,A -85,B 0,C 180,E1 28789.915,E2 28789.915} C_VEL
LIN {X 0,Y 656.679,Z 491.422,A -85,B 0,C 180,E1 28786.976,E2 28786.976} C_VEL
LIN {X 0,Y 656.673,Z 491.42,A -85,B 0,C 180,E1 28783.73,E2 28783.73} C_VEL
LIN {X 0,Y 656.678,Z 491.432,A -85,B 0,C 180,E1 28780.798,E2 28780.798} C_VEL
LIN {X 0,Y 656.672,Z 491.427,A -85,B 0,C 180,E1 28777.552,E2 28777.552} C_VEL
LIN {X 0,Y 656.672,Z 491.423,A -85,B 0,C 180,E1 28774.667,E2 28774.667} C_VEL
LIN {X 0,Y 656.676,Z 491.422,A -85,B 0,C 180,E1 28771.438,E2 28771.438} C_VEL
LIN {X 0,Y 656.661,Z 491.43,A -85,B 0,C 180,E1 28768.617,E2 28768.617} C_VEL
LIN {X 0,Y 656.693,Z 491.413,A -85,B 0,C 180,E1 28765.457,E2 28765.457} C_VEL
LIN {X 0,Y 656.654,Z 491.431,A -85,B 0,C 180,E1 28762.587,E2 28762.587} C_VEL
LIN {X 0,Y 656.712,Z 491.415,A -85,B 0,C 180,E1 28759.562,E2 28759.562} C_VEL
LIN {X 0,Y 656.649,Z 491.408,A -85,B 0,C 180,E1 28756.578,E2 28756.578} C_VEL
LIN {X 0,Y 656.709,Z 491.421,A -85,B 0,C 180,E1 28753.607,E2 28753.607} C_VEL
LIN {X 0,Y 656.738,Z 491.611,A -85,B 0,C 180,E1 28751.396,E2 28751.396} C_VEL
LIN {X 0,Y 659.276,Z 498.11,A -85,B 0,C 180,E1 28750.703,E2 28750.703} C_VEL
LIN {X 0,Y 667.11,Z 516.607,A -85,B 0,C 180,E1 28748.863,E2 28748.863} C_VEL
LIN {X 0,Y 670.039,Z 524.284,A -85,B 0,C 180,E1 28748.146,E2 28748.146} C_VEL
LIN {X 0,Y 669.852,Z 531.933,A -85,B 0,C 180,E1 28747.682,E2 28747.682} C_VEL
LIN {X 0,Y 673.42,Z 549.93,A -85,B 0,C 180,E1 28747.241,E2 28747.241} C_VEL
LIN {X 0,Y 671.242,Z 791.049,A -85,B 0,C 180,E1 28744.362,E2 28744.362} C_VEL
LIN {X 0,Y 670.227,Z 914.657,A -85,B 0,C 180,E1 28742.915,E2 28742.915} C_VEL
LIN {X 0,Y 669.7,Z 937.495,A -85,B 0,C 180,E1 28742.541,E2 28742.541} C_VEL
LIN {X 0,Y 668.852,Z 962.038,A -85,B 0,C 180,E1 28741.976,E2 28741.976} C_VEL
LIN {X 0,Y 668.075,Z 981.319,A -85,B 0,C 180,E1 28741.413,E2 28741.413} C_VEL
LIN {X 0,Y 667.055,Z 1003.447,A -85,B 0,C 180,E1 28740.637,E2 28740.637} C_VEL
LIN {X 0,Y 665.827,Z 1026.274,A -85,B 0,C 180,E1 28739.657,E2 28739.657} C_VEL
LIN {X 0,Y 664.639,Z 1047.752,A -85,B 0,C 180,E1 28738.58,E2 28738.58} C_VEL
LIN {X 0,Y 663.3,Z 1069.069,A -85,B 0,C 180,E1 28737.323,E2 28737.323} C_VEL
LIN {X 0,Y 662.101,Z 1089.076,A -85,B 0,C 180,E1 28735.972,E2 28735.972} C_VEL
LIN {X 0,Y 660.891,Z 1108.081,A -85,B 0,C 180,E1 28734.49,E2 28734.49} C_VEL
LIN {X 0,Y 659.869,Z 1125.394,A -85,B 0,C 180,E1 28732.965,E2 28732.965} C_VEL
LIN {X 0,Y 658.885,Z 1142.257,A -85,B 0,C 180,E1 28731.265,E2 28731.265} C_VEL
LIN {X 0,Y 658.101,Z 1157.482,A -85,B 0,C 180,E1 28729.527,E2 28729.527} C_VEL
LIN {X 0,Y 657.381,Z 1171.986,A -85,B 0,C 180,E1 28727.618,E2 28727.618} C_VEL
LIN {X 0,Y 656.887,Z 1183.989,A -85,B 0,C 180,E1 28725.811,E2 28725.811} C_VEL
LIN {X 0,Y 656.474,Z 1195.728,A -85,B 0,C 180,E1 28723.745,E2 28723.745} C_VEL
LIN {X 0,Y 656.243,Z 1204.375,A -85,B 0,C 180,E1 28721.959,E2 28721.959} C_VEL
LIN {X 0,Y 656.044,Z 1213.3,A -85,B 0,C 180,E1 28719.74,E2 28719.74} C_VEL
LIN {X 0,Y 655.955,Z 1219.237,A -85,B 0,C 180,E1 28717.885,E2 28717.885} C_VEL
LIN {X 0,Y 655.934,Z 1224.338,A -85,B 0,C 180,E1 28715.862,E2 28715.862} C_VEL
LIN {X 0,Y 655.912,Z 1227.898,A -85,B 0,C 180,E1 28713.758,E2 28713.758} C_VEL
LIN {X 0,Y 655.902,Z 1229.835,A -85,B 0,C 180,E1 28711.834,E2 28711.834} C_VEL
LIN {X 0,Y 655.885,Z 1230.395,A -85,B 0,C 180,E1 28709.563,E2 28709.563} C_VEL
LIN {X 0,Y 655.914,Z 1229.498,A -85,B 0,C 180,E1 28707.729,E2 28707.729} C_VEL
LIN {X 0,Y 655.922,Z 1226.916,A -85,B 0,C 180,E1 28705.536,E2 28705.536} C_VEL
LIN {X 0,Y 655.938,Z 1222.896,A -85,B 0,C 180,E1 28703.523,E2 28703.523} C_VEL
LIN {X 0,Y 656.003,Z 1217.694,A -85,B 0,C 180,E1 28701.58,E2 28701.58} C_VEL
LIN {X 0,Y 656.121,Z 1210.075,A -85,B 0,C 180,E1 28699.404,E2 28699.404} C_VEL
LIN {X 0,Y 656.29,Z 1202.28,A -85,B 0,C 180,E1 28697.581,E2 28697.581} C_VEL
LIN {X 0,Y 656.62,Z 1191.384,A -85,B 0,C 180,E1 28695.448,E2 28695.448} C_VEL
LIN {X 0,Y 657.022,Z 1180.553,A -85,B 0,C 180,E1 28693.648,E2 28693.648} C_VEL
LIN {X 0,Y 657.642,Z 1166.732,A -85,B 0,C 180,E1 28691.656,E2 28691.656} C_VEL
LIN {X 0,Y 658.319,Z 1152.859,A -85,B 0,C 180,E1 28689.925,E2 28689.925} C_VEL
LIN {X 0,Y 659.237,Z 1136.167,A -85,B 0,C 180,E1 28688.093,E2 28688.093} C_VEL
LIN {X 0,Y 660.181,Z 1119.822,A -85,B 0,C 180,E1 28686.527,E2 28686.527} C_VEL
LIN {X 0,Y 661.337,Z 1101.299,A -85,B 0,C 180,E1 28684.955,E2 28684.955} C_VEL
LIN {X 0,Y 662.477,Z 1082.415,A -85,B 0,C 180,E1 28683.562,E2 28683.562} C_VEL
LIN {X 0,Y 663.804,Z 1061.606,A -85,B 0,C 180,E1 28682.213,E2 28682.213} C_VEL
LIN {X 0,Y 664.992,Z 1040.827,A -85,B 0,C 180,E1 28681.058,E2 28681.058} C_VEL
LIN {X 0,Y 666.289,Z 1018.504,A -85,B 0,C 180,E1 28679.986,E2 28679.986} C_VEL
LIN {X 0,Y 667.354,Z 996.997,A -85,B 0,C 180,E1 28679.126,E2 28679.126} C_VEL
LIN {X 0,Y 668.265,Z 976.882,A -85,B 0,C 180,E1 28678.447,E2 28678.447} C_VEL
LIN {X 0,Y 669.206,Z 951.359,A -85,B 0,C 180,E1 28677.757,E2 28677.757} C_VEL
LIN {X 0,Y 669.903,Z 929.612,A -85,B 0,C 180,E1 28677.316,E2 28677.316} C_VEL
LIN {X 0,Y 670.462,Z 900.182,A -85,B 0,C 180,E1 28676.901,E2 28676.901} C_VEL
LIN {X 0,Y 672.258,Z 661.55,A -85,B 0,C 180,E1 28674.113,E2 28674.113} C_VEL
LIN {X 0,Y 673.262,Z 548.149,A -85,B 0,C 180,E1 28672.727,E2 28672.727} C_VEL
LIN {X 0,Y 669.763,Z 531.386,A -85,B 0,C 180,E1 28672.302,E2 28672.302} C_VEL
LIN {X 0,Y 669.957,Z 523.576,A -85,B 0,C 180,E1 28671.801,E2 28671.801} C_VEL
LIN {X 0,Y 660.933,Z 501.863,A -85,B 0,C 180,E1 28669.683,E2 28669.683} C_VEL
LIN {X 0,Y 656.768,Z 491.792,A -85,B 0,C 180,E1 28668.64,E2 28668.64} C_VEL
LIN {X 0,Y 656.668,Z 491.4,A -85,B 0,C 180,E1 28668.054,E2 28668.054} C_VEL
LIN {X 0,Y 656.66,Z 491.426,A -85,B 0,C 180,E1 28665.201,E2 28665.201} C_VEL
LIN {X 0,Y 656.689,Z 491.428,A -85,B 0,C 180,E1 28662.011,E2 28662.011} C_VEL
LIN {X 0,Y 656.651,Z 491.399,A -85,B 0,C 180,E1 28659.192,E2 28659.192} C_VEL
LIN {X 0,Y 656.709,Z 491.43,A -85,B 0,C 180,E1 28656.202,E2 28656.202} C_VEL
LIN {X 0,Y 656.653,Z 491.4,A -85,B 0,C 180,E1 28653.242,E2 28653.242} C_VEL
LIN {X 0,Y 656.714,Z 491.425,A -85,B 0,C 180,E1 28650.263,E2 28650.263} C_VEL
LIN {X 0,Y 656.663,Z 491.432,A -85,B 0,C 180,E1 28647.181,E2 28647.181} C_VEL
LIN {X 0,Y 656.701,Z 491.417,A -85,B 0,C 180,E1 28644.216,E2 28644.216} C_VEL
LIN {X 0,Y 656.672,Z 491.424,A -85,B 0,C 180,E1 28641.154,E2 28641.154} C_VEL
LIN {X 0,Y 656.688,Z 491.425,A -85,B 0,C 180,E1 28638.179,E2 28638.179} C_VEL
LIN {X 0,Y 656.676,Z 491.432,A -85,B 0,C 180,E1 28635.002,E2 28635.002} C_VEL
LIN {X 0,Y 656.684,Z 491.417,A -85,B 0,C 180,E1 28632.04,E2 28632.04} C_VEL
LIN {X 0,Y 656.677,Z 491.42,A -85,B 0,C 180,E1 28628.823,E2 28628.823} C_VEL
LIN {X 0,Y 656.687,Z 491.424,A -85,B 0,C 180,E1 28625.855,E2 28625.855} C_VEL
LIN {X 0,Y 656.68,Z 491.429,A -85,B 0,C 180,E1 28622.618,E2 28622.618} C_VEL
LIN {X 0,Y 656.691,Z 491.42,A -85,B 0,C 180,E1 28619.651,E2 28619.651} C_VEL
LIN {X 0,Y 656.68,Z 491.431,A -85,B 0,C 180,E1 28616.421,E2 28616.421} C_VEL
LIN {X 0,Y 656.702,Z 491.416,A -85,B 0,C 180,E1 28613.355,E2 28613.355} C_VEL
LIN {X 0,Y 656.677,Z 491.42,A -85,B 0,C 180,E1 28610.181,E2 28610.181} C_VEL
LIN {X 0,Y 656.704,Z 491.424,A -85,B 0,C 180,E1 28607.156,E2 28607.156} C_VEL
LIN {X 0,Y 656.681,Z 491.432,A -85,B 0,C 180,E1 28604.002,E2 28604.002} C_VEL
LIN {X 0,Y 656.703,Z 491.415,A -85,B 0,C 180,E1 28600.984,E2 28600.984} C_VEL
LIN {X 0,Y 656.682,Z 491.423,A -85,B 0,C 180,E1 28597.814,E2 28597.814} C_VEL
LIN {X 0,Y 656.707,Z 491.424,A -85,B 0,C 180,E1 28594.74,E2 28594.74} C_VEL
LIN {X 0,Y 656.684,Z 491.432,A -85,B 0,C 180,E1 28591.636,E2 28591.636} C_VEL
LIN {X 0,Y 656.708,Z 491.423,A -85,B 0,C 180,E1 28588.619,E2 28588.619} C_VEL
